// ---- Library/10_Machine/11_IOData/GVL_Output.TcGVL
{attribute 'qualified_only'}
VAR_GLOBAL
	uniDO : uni_OutputModule;
END_VAR

// ---- Library/10_Machine/12_MachineControl/GVL_Machine.TcGVL
VAR_GLOBAL
    PackTags               : ARRAY[0..3] OF ST_PackMLv30; //PackTags
    bButtonProductionReq   : BOOL; //TRUE when a mode change to PRODUCTION is requested
    stChangeIntoProduction : ST_ChangeIntoProduction; //Result of command box "Change to Production requested"
    CylinderStatus         : ST_CylinderStatus;
    RemoteData             : ST_SetupPara;
    AllocatYAxisHome       : BOOL;
END_VAR
VAR_GLOBAL PERSISTENT
    LocalData : ST_SetupPara;
END_VAR

// ---- Library/10_Machine/12_MachineControl/GVL_Machine_Const.TcGVL
VAR_GLOBAL CONSTANT
	udiMax_CylinderNum : UDINT := 53;
END_VAR

// ---- Library/10_Machine/18_HMI_Handshake/GVL_ADS.TcGVL
{attribute 'qualified_only'}
VAR_GLOBAL
	StorageTask 		:   E_MachineTask;
	NeedleTask			:   E_MachineTask;
	ShippingTask		:   E_MachineTask;
	
	PCTask              :  	ST_PCTask;
	//手動模式
	Manualmode			:	ST_MachineAdjust;
	//自動
 	Automode 			:	ST_MachineTask;   
	ActiveFinishing 	:	ST_ActiveResult;
	MachineMode         :   ST_Mode;
	
END_VAR

// ---- Library/10_Machine/18_HMI_Handshake/GVL_HMI.TcGVL
{attribute 'qualified_only'}
VAR_GLOBAL
    ControlOutPut 	: ST_HMI_ControlOutPut;//手臂以及馬達動作命令
    ControlConvery  : ST_HMI_ControlConvery;//軌道動作命令
    ControlInPut 	: ST_HMI_ControlInPut;//X點位
    Setup     		: ST_SetupPara;//參數
    Status    		: ST_HMI_MachineStatus;//狀態
END_VAR

// ---- POUs/ModbusRTU/00_BaseFBs/01_FB_ObjectBase/GVLs/Para_ObjectBase.TcGVL
{attribute 'qualified_only'}
VAR_GLOBAL CONSTANT
	cNumCmdRecord			: UINT := 500;
	cNumMsgRecord			: UINT := 1000;
END_VAR

// ---- Library/00_PackML/01_ObjectBase/I_ErrorElement.TcIO
INTERFACE I_ErrorElement

METHOD M_GetError
VAR_INPUT
END_VAR
VAR_OUTPUT
	Error : BOOL;
	ErrorID : DINT;
	ErrorMsg : T_MaxString;
END_VAR
END_METHOD

METHOD M_GetName :STRING
VAR_INPUT
END_VAR
END_METHOD

METHOD RegisterAlarm
VAR_INPUT
	Trigger : REFERENCE TO BOOL;
	ID : DINT;
	value :DINT;
	Message : STRING;
	Category : DINT;
END_VAR
END_METHOD

END_INTERFACE

// ---- Library/00_PackML/01_ObjectBase/I_ErrorSubject.TcIO
INTERFACE I_ErrorSubject

END_INTERFACE

// ---- POUs/ModbusRTU/00_BaseFBs/01_FB_ObjectBase/ITFs/IBasicElement.TcIO
INTERFACE IBasicElement

METHOD GetModelState
VAR_INPUT
END_VAR
VAR_OUTPUT
    xDone : BOOL;
    xBusy : BOOL;
    xError : BOOL;
    xAborted : BOOL;
    iErrorID : UDINT;
	UniqueErrorCode : STRING;
END_VAR
END_METHOD

METHOD GetName : STRING
VAR_INPUT
END_VAR
END_METHOD

END_INTERFACE

// ---- POUs/ModbusRTU/ComModbusRTU.TcPOU
PROGRAM ComModbusRTU
VAR
	MB_EL6X22B_ControllerN				:	ARRAY[0..3] OF ModbusRtuMasterV2_KL6x22B;
	MBUnusedData_Read 					: 	ARRAY[0..3] OF ARRAY[0..7] OF BYTE;
	MBSensorError_Read 					: 	ARRAY[0..3] OF ARRAY[0..21] OF BYTE;
	nErrID_ControllerN					:	ARRAY[0..3] OF MODBUS_ERRORS;
	iReadMBAddr							:	ARRAY[0..3] OF WORD;
	bBusy_ControllerN					:	ARRAY[0..3] OF BOOL;
	bError_ControllerN					:	ARRAY[0..3] OF BOOL;
	fbComReset_ControllerN				:	ARRAY[0..3] OF ComReset;
	bComReset							:	ARRAY[0..3] OF BOOL;
	bComResetBusy							:	ARRAY[0..3] OF BOOL;
	bComResetError							:	ARRAY[0..3] OF BOOL;
	bStart								:	ARRAY[0..3] OF BOOL;
	
	actStart							:	ARRAY[0..3] OF ULINT;
	actEnd								:	ARRAY[0..3] OF ULINT;
	exeTime								:	ARRAY[0..3] OF ULINT;
	nSlave								:	BYTE;
	MBdata_Read_ControllerN	 AT %I*		: 	ARRAY[0..3] OF ARRAY[0..21] OF BYTE;
	bMasterError						:	ARRAY[0..3] OF BOOL;
	nStep								:	UINT;
	bModbusRTUError						:	BOOL;
	udiModbusRTUErrorID					:	UDINT;
	nAlias								:	UINT;
	bPassModBusMaster					:	ARRAY[0..3] OF BOOL;
	
	
	//================Alternative======================
	//fb_Warehouse_Modbus :ARRAY[0..3] OF FB_CommunicateModbusRTU; //0&1 : warehouse A , 2&3 : warehouse B
		//Declared in GVL due to Error handling request
	I		:UINT;
	SensorState	: ARRAY[0..99] OF BOOL;
	SensorStatesAll : un_RS485States_all;
	arr485sensor					: ARRAY [0..399] OF BOOL;
	fb_Warehouse_Modbus : ARRAY [0..3] OF FB_CommunicateModbusRTU;
	bMotorCoreUpdated	:	BOOL := TRUE;
	bReset				:	BOOL;
END_VAR

//M_CommunicateModbusRTU(bReset:=GVL.Reset,
//						bModBusRTUError=>bModbusRTUError,
//						udiModbusRTUErrorID=>udiModbusRTUErrorID);
						
//GVL.fbModbusRTUErrorTrans(
//	xDone:= , 
//	xBusy:= , 
//	xError:= bModbusRTUError, 
//	xAborted:= , 
//	iErrorID:= udiModbusRTUErrorID, 
//	Name:= 'Communicate ModBus RTU ');
	
	
	
//=================Alternative======================================

//Update FBs
FOR I :=0 TO 3 BY 1 DO
	fb_Warehouse_Modbus[I](Execute:=bMotorCoreUpdated AND NOT bPassModBusMaster[I] , 
							   unitID :=UINT_TO_BYTE(I)+1 , 
							   Reset:=bReset,
							   MBdata_Read_ControllerN :=MBdata_Read_ControllerN[I],
							   ObjectName:=CONCAT('Communicate ModBus RTU : ',UINT_TO_STRING(I)),
							   arrSensor=>SensorStatesAll.arrSensorByController[I]);
	
	arr485sensor := SensorStatesAll.arrSensorAll;
	
END_FOR


//bPassModBusMaster[0] := GVL.stModbusByPass.switchOff_1;
//bPassModBusMaster[1] := GVL.stModbusByPass.switchOff_2;
//bPassModBusMaster[2] := GVL.stModbusByPass.switchOff_3;
//bPassModBusMaster[3] := GVL.stModbusByPass.switchOff_4;

END_PROGRAM

// ---- POUs/ModbusRTU/SerialComTask/FB_CommunicateModbusRTU.TcPOU
FUNCTION_BLOCK FB_CommunicateModbusRTU EXTENDS FB_ObjectBase_V2
VAR_INPUT
//    Execute    :BOOL;   // True : This prog will start.
//    Abort      :BOOL;   // True : This prog will be abort.
//    Reset      :BOOL;   // True : This prog will be reset.
//    ObjectName :STRING; // Set this fb name(About it's action)
	  
	  
	  unitID	  :BYTE;
	  MBdata_Read_ControllerN	: REFERENCE TO 	ARRAY[0..21] OF BYTE;
END_VAR

VAR_OUTPUT
//    Busy    :BOOL;        // True : This prog is running.
//    Done    :BOOL;        // True : Command has been executed.
//    Aborted :BOOL;        // True : This prog is aborted.
//    Error   :BOOL;        // True : This prog has an error.
//    ErrorID :UINT;       // Output ErrorID
//    Status  :T_MaxString; // Output this prog status by string(255bytes)
	arrSensor		: ARRAY[0..99] OF BOOL;
END_VAR

VAR
//    eState :E_MethodStatus_Basic;
//	uiExecutingStep : UDINT; // This var is used to been controll STATE_EXECUTING process.
//	uiResettingStep : UDINT;
//	uiAbortingStep : UDINT;
//	_Executed :BOOL; // Executing process completed.
//	_Error : BOOL; // FB has an error.
//	_ResetCompleted : BOOL; // FB resetting completed.
//	_AbortCompleted : BOOL; // FB aborting completed.
	_Abort		: BOOL;
	strStatus	: STRING;
	uiResumeStep : UINT;
	arrSensorEmpty : ARRAY[0..99] OF BOOL;
	MB_EL6X22B_ControllerN	: ModbusRtuMasterV2_KL6x22B;
	fbComReset_ControllerN	: ComReset;	
	fbClearComBuffer		: ClearComBuffer;
	SensorState : un_RS485States;
	bComReset	:BOOL;
	bComResetBusy :BOOL;
	bComResetError :BOOL;
	bFB_ErrorOccur :BOOL;
END_VAR

A00_BasicUnits();
SUPER^.A10_StateControl();

ACTION A00_BasicUnits:
MB_EL6X22B_ControllerN();
fbComReset_ControllerN(
		Execute:= bComReset, 
		pComIn:= ADR(MB_EL6X22B_ControllerN.InData), 
		pComOut:= ADR(MB_EL6X22B_ControllerN.OutData), 
		SizeComIn:= SIZEOF(MB_EL6X22B_ControllerN.InData), 
		Done=> , 
		Busy=> bComResetBusy, 
		Error=> bComResetError, 
		ErrorID=> );
END_ACTION

METHOD GetModelState
VAR_OUTPUT
    xDone    :BOOL;
    xBusy    :BOOL;
    xError   :BOOL;
    xAborted :BOOL;
    iErrorID :UDINT;
	UniqueErrorCode : STRING;
END_VAR
xDone    := Done;
xBusy    := Busy;
xError   := Error;
xAborted := Abort;
iErrorID := ErrorID;
END_METHOD

METHOD GetName : STRING
GetName := ObjectName;
END_METHOD

METHOD PRIVATE M_AnalyzeData : BOOL
VAR_INPUT
	Data : ARRAY [0..21] OF BYTE;
END_VAR

VAR_OUTPUT
	arrSensor : ARRAY[0..9] OF BOOL;
END_VAR

arrSensor[0] :=Data[4].1;
arrSensor[1] :=Data[4].0;
arrSensor[2] :=Data[3].7;
arrSensor[3] :=Data[3].6;
arrSensor[4] :=Data[3].5;
arrSensor[5] :=Data[3].4;
arrSensor[6] :=Data[3].3;
arrSensor[7] :=Data[3].2;
arrSensor[8] :=Data[3].1;
arrSensor[9] :=Data[3].0;
END_METHOD

METHOD  M_STATE_ABORTED
VAR_INPUT
END_VAR
ERROR :=TRUE;
Busy    := FALSE;
Aborted := TRUE;
Status := strStatus;

IF NOT Execute THEN
	eSTATE:=STATE_RESETTING;
END_IF

IF Execute AND Reset THEN
	uiExecutingStep :=uiResumeStep;
	eSTATE:=STATE_EXECUTING;
END_IF
END_METHOD

METHOD  M_STATE_ABORTING
VAR_INPUT
END_VAR
CASE uiAbortingStep OF
	0 :
		uiAbortingStep:=9999;
	
	9999:	_AbortCompleted:=TRUE;
END_CASE

IF _AbortCompleted THEN	
	eSTATE :=STATE_ABORTED;
END_IF
END_METHOD

METHOD  M_STATE_DONE
VAR_INPUT
END_VAR
Busy 	:= FALSE;
Done	:=TRUE;

IF NOT Execute THEN
	eSTATE:=STATE_RESETTING;
END_IF
END_METHOD

METHOD  M_STATE_DORMANT
VAR_INPUT
END_VAR
Busy            := FALSE;
Done            := FALSE;
Aborted         := FALSE;
Error           := FALSE;
ErrorID         := 0;
Status          := '';
_ResetCompleted := FALSE;
_Error          := FALSE;
_Executed       := FALSE;
strStatus :='No Error';
uiExecutingStep :=uiResettingStep :=uiResumeStep :=0;
bComReset		:= FALSE;

arrSensor :=arrSensorEmpty;
// output all false if program stop working

IF Execute THEN
	eSTATE:=STATE_EXECUTING;
END_IF
END_METHOD

METHOD  M_STATE_ERROR
VAR_INPUT
END_VAR

VAR
	tempStr	:	STRING ;
END_VAR
ERROR   :=TRUE;
Busy	:=FALSE;
tempStr := CONCAT( 'Controllor ' , BYTE_TO_STRING(unitID));
Status := CONCAT(tempStr, strStatus);
ErrorID := unitID + 2600;// Start from 2600

IF NOT Execute OR Reset	THEN	
	eSTATE:=STATE_RESETTING;
END_IF
END_METHOD

METHOD  M_STATE_EXECUTING
VAR_INPUT
END_VAR

VAR
	arrSensorSingleModule : ARRAY [0..9] OF BOOL;	
	pMemoryAddr : ARRAY[0..7] OF BYTE;
END_VAR

VAR_INST
	Quantity : WORD;
	cbLength : UINT;
	
	iReadMBAddr :  WORD :=0;
END_VAR
Busy :=TRUE;
IF  MB_EL6X22B_ControllerN.Error AND NOT bFB_ErrorOccur  THEN
	bFB_ErrorOccur :=TRUE;
	_Error :=TRUE;
	strStatus :=' Modbus connection error';
END_IF

arrSensor:=SensorState.arrSensorByController;

IF iReadMBAddr <= 900 THEN
		Quantity :=10;	
	    cbLength :=20;
		MB_EL6X22B_ControllerN.ReadCoils();
ELSE
		Quantity :=1;
		cbLength :=2;
		MB_EL6X22B_ControllerN.ReadInputRegs();
END_IF

CASE uiExecutingStep OF
	
0: // Init
	MB_EL6X22B_ControllerN.Execute:=FALSE;
	iReadMBAddr:=0;
	uiExecutingStep:=100;
	
100:	
	MB_EL6X22B_ControllerN.UnitID:= unitID;
	MB_EL6X22B_ControllerN.Quantity:= Quantity; 
	MB_EL6X22B_ControllerN.MBAddr:= iReadMBAddr; 
	MB_EL6X22B_ControllerN.cbLength:= cbLength;
	MB_EL6X22B_ControllerN.pMemoryAddr:=ADR(pMemoryAddr) ; 
	MB_EL6X22B_ControllerN.Timeout:= T#1000MS; 
	MB_EL6X22B_ControllerN.Execute:=TRUE;	
	IF MB_EL6X22B_ControllerN.BUSY THEN
		uiExecutingStep:=200;
	END_IF	
	IF bFB_ErrorOccur THEN
		uiExecutingStep:=110;		
	END_IF
	
110:
	bFB_ErrorOccur :=FALSE; //Internal error flag 
	IF MB_EL6X22B_ControllerN.BUSY THEN
		uiExecutingStep:=200;
	END_IF
		
200:
	IF NOT MB_EL6X22B_ControllerN.BUSY THEN
		MB_EL6X22B_ControllerN.Execute:=FALSE;
		
		IF iReadMBAddr>=1000 THEN
			// Error checking step			
			IF MBdata_Read_ControllerN[1] = 4 AND MBdata_Read_ControllerN[3] + MBdata_Read_ControllerN[4] > 0 THEN
				_Error := TRUE;
				strStatus :=' Controller report error';
			END_IF
			
			iReadMBAddr :=0;
			
		ELSE
			// Signal step
			M_AnalyzeData(Data :=MBdata_Read_ControllerN,arrSensor=>arrSensorSingleModule);
			SensorState.arrSensorBySingleModule[iReadMBAddr/100] :=arrSensorSingleModule;		
			iReadMBAddr :=iReadMBAddr +100;
		END_IF
		
		uiExecutingStep:=100;		
		
	 END_IF

END_CASE
	
IF NOT Execute THEN
	eState:=STATE_RESETTING;
END_IF
IF _Error THEN
	eState:=STATE_ERROR;
END_IF
IF _Abort THEN
	eSTATE:=STATE_ABORTING;
END_IF
IF _Executed THEN
	eSTATE:=STATE_Done;
END_IF
END_METHOD

METHOD  M_STATE_RESETTING
VAR_INPUT
END_VAR
Error :=FALSE;
Done :=FALSE;
Busy := FALSE;


CASE uiResettingStep OF
	
	0:
		MB_EL6X22B_ControllerN.Execute:=FALSE;
//		fbClearComBuffer(Buffer:=MB_EL6X22B_ControllerN.InData);
//		fbClearComBuffer(Buffer:=MB_EL6X22B_ControllerN.OutData);
		uiResettingStep:=100;
	100:	
		bComReset := TRUE;
		IF fbComReset_ControllerN.Busy THEN
			uiResettingStep:=200;
		END_IF
	200:
		IF fbComReset_ControllerN.Done THEN
			uiResettingStep:=9999;
		END_IF

	9999:
		_Error:=FALSE;
		_ResetCompleted:=TRUE;
END_CASE
IF _ResetCompleted THEN
	eSTATE:=STATE_DORMANT;
END_IF
END_METHOD

END_FUNCTION_BLOCK

// ---- POUs/ModbusRTU/00_BaseFBs/01_FB_ObjectBase/FB_ObjectBase_V2.TcPOU
FUNCTION_BLOCK FB_ObjectBase_V2 IMPLEMENTS IBasicElement
VAR_INPUT
    Execute    :BOOL;   // True : This prog will start.
    Abort      :BOOL;   // True : This prog will be abort.
    Reset      :BOOL;   // True : This prog will be reset.
    ObjectName :STRING; // Set this fb name(About it's action)
END_VAR

VAR_OUTPUT
    Busy    :BOOL;        // True : This prog is running.
    Done    :BOOL;        // True : Command has been executed.
    Aborted :BOOL;        // True : This prog is aborted.
    Error   :BOOL;        // True : This prog has an error.
    ErrorID :UINT;       // Output ErrorID
    Status  :STRING; // Output this prog status by string(255bytes)
	UniqueErrorCode :STRING;	
END_VAR

VAR
    eState :E_MethodStatus_Basic;
	uiExecutingStep : UDINT; // This var is used to been controll STATE_EXECUTING process.
	uiResettingStep : UDINT;
	uiAbortingStep : UDINT;
	_Executed :BOOL; // Executing process completed.
	_Error : BOOL; // FB has an error.
	_ResetCompleted : BOOL; // FB resetting completed.
	_AbortCompleted : BOOL; // FB aborting completed.
END_VAR

A00_BasicUnits();
A10_StateControl();

ACTION A00_BasicUnits:

END_ACTION

ACTION A10_StateControl:
CASE eState OF
	STATE_DORMANT:
		M_STATE_DORMANT();
	STATE_EXECUTING:
		M_STATE_EXECUTING();
	STATE_ABORTING:
		M_STATE_ABORTING();
	STATE_ABORTED:
		M_STATE_ABORTED();
	STATE_DONE:
		M_STATE_DONE();
	STATE_ERROR:
		M_STATE_ERROR();
	STATE_RESETTING:
		M_STATE_RESETTING();
END_CASE
END_ACTION

METHOD GetModelState
VAR_OUTPUT
    xDone    :BOOL;
    xBusy    :BOOL;
    xError   :BOOL;
    xAborted :BOOL;
    iErrorID :UDINT;	
	UniqueErrorCode : STRING;
END_VAR
xDone    := Done;
xBusy    := Busy;
xError   := Error;
xAborted := Abort;
iErrorID := ErrorID;
UniqueErrorCode := THIS^.UniqueErrorCode;
END_METHOD

METHOD GetName : STRING
GetName := ObjectName;
END_METHOD

METHOD M_RefLinks
VAR_INPUT
END_VAR
END_METHOD

METHOD  M_STATE_ABORTED
VAR_INPUT
END_VAR
;
END_METHOD

METHOD  M_STATE_ABORTING
VAR_INPUT
END_VAR
;
END_METHOD

METHOD  M_STATE_DONE
VAR_INPUT
END_VAR
;
END_METHOD

METHOD  M_STATE_DORMANT
VAR_INPUT
END_VAR
;
END_METHOD

METHOD  M_STATE_ERROR
VAR_INPUT
END_VAR
;
END_METHOD

METHOD  M_STATE_EXECUTING
VAR_INPUT
END_VAR
;
END_METHOD

METHOD  M_STATE_RESETTING
VAR_INPUT
END_VAR
;
END_METHOD

END_FUNCTION_BLOCK

// ---- POUs/DAS_CoreSys.TcPOU
PROGRAM DAS_CoreSys
VAR
    UserModeCofig  : PML_UnitModeConfig; //User can configure his own Mode
    MachineControl : FB_MachineControl;
	CoreSys_Stop : BOOL;
	CoreSys_Reset :BOOL;
	CoreSys_Start : BOOL;
	CoreSys_Estop : BOOL;
	OP_Mode : E_UnitMode := E_UnitMode.Manual;
END_VAR

A00_BasicUnit();
A10_StatusCtrl();


CASE GVL_ADS.MachineMode.TargetMode OF
		E_MachineMode.MANUAL:
			OP_Mode := E_UnitMode.Manual;
		E_MachineMode.AUTO:
			OP_Mode := E_UnitMode.Auto;
ELSE
	OP_Mode := E_UnitMode.Manual;
END_CASE
IF OP_Mode = E_UnitMode.Manual THEN
	GVL_ADS.MachineMode.CurrentMode := E_MachineMode.MANUAL;
ELSIF OP_Mode = E_UnitMode.Auto THEN
	GVL_ADS.MachineMode.CurrentMode := E_MachineMode.AUTO;
END_IF

ACTION A00_BasicUnit:
CoreSys_Start := MachineControl.Machine_Start;
CoreSys_Stop := MachineControl.Machine_Stop;
CoreSys_Reset := MachineControl.Machine_Reset;
MachineControl(
    eModeCommand := PackTags[0].Command.UnitMode,
    eStateCommand := PackTags[0].Command.CntrlCmd,
    PackTag := PackTags[0],
    INPUT := GVL_Input.uniDI.stDI,
    OUTPUT := GVL_Output.uniDO.stDO); // FB_MachineControl
PackTags[0].Status.StateCurrent := MachineControl.eStateCurrent;
PackTags[0].Status.UnitModeCurrent := MachineControl.eModeCurrent;
CoreSys_Estop := MachineControl.Machine_Estop;
END_ACTION

ACTION A01_UnitModeConfig:
//UserModeCofig(
//	eMode							:= ePMLUnitMode_Service, 
//	bDisableClearing				:= TRUE, 
//	bDisableStarting				:= TRUE, 
//	bDisableSuspended				:= FALSE, 
//	bDisableStopping				:= TRUE, 
//	bDisableAborting				:= TRUE, 
//	bDisableHolding					:= TRUE, 
//	bDisableHeld					:= TRUE, 
//	bDisableUnholding				:= TRUE, 
//	bDisableSuspending				:= TRUE, 
//	bDisableUnsuspending			:= TRUE, 
//	bDisableResetting				:= TRUE, 
//	bDisableIdle					:= TRUE, 
//	bDisableCompleting				:= TRUE, 
//	bDisableComplete				:= TRUE, 
//	bEnableUnitModeChangeStopped	:= TRUE, 
//	bEnableUnitModeChangeIdle		:= FALSE, 
//	bEnableUnitModeChangeSuspended	:= FALSE, 
//	bEnableUnitModeChangeExecute	:= FALSE, 
//	bEnableUnitModeChangeAborted	:= TRUE, 
//	bEnableUnitModeChangeHeld		:= FALSE, 
//	bEnableUnitModeChangeComplete	:= FALSE, 
//	bError							=> , 
//	nErrorId						=> );
END_ACTION

ACTION A10_StatusCtrl:
IF PackTags[0].Status.UnitModeCurrent = E_UnitMode.Manual THEN
	IF PackTags[0].Status.StateCurrent = ePMLState_Aborted AND NOT MachineControl.Error THEN
		PackTags[0].Command.CntrlCmd := ePMLCommand_Clear;
	END_IF
	IF PackTags[0].Status.StateCurrent = ePMLState_Stopped THEN
		IF OP_Mode = E_UnitMode.Manual THEN
		PackTags[0].Command.CntrlCmd := ePMLCommand_Reset;
		END_IF
	END_IF
	IF PackTags[0].Status.StateCurrent = ePMLState_Idle THEN
		PackTags[0].Command.CntrlCmd := ePMLCommand_Start;
	END_IF
ELSIF PackTags[0].Status.UnitModeCurrent = E_UnitMode.Auto THEN
	IF PackTags[0].Status.StateCurrent = ePMLState_Aborted AND NOT MachineControl.Error THEN
		PackTags[0].Command.CntrlCmd := ePMLCommand_Clear;
	END_IF
	IF PackTags[0].Status.StateCurrent = ePMLState_Stopped THEN
		IF OP_Mode = E_UnitMode.Auto THEN
		PackTags[0].Command.CntrlCmd := ePMLCommand_Reset;
		END_IF
	END_IF
	IF PackTags[0].Status.StateCurrent = ePMLState_Idle THEN
		PackTags[0].Command.CntrlCmd := ePMLCommand_Start;
	END_IF
END_IF

IF PackTags[0].Status.UnitModeCurrent = E_UnitMode.Manual THEN
    IF ((PackTags[0].Status.StateCurrent = ePMLState_Stopped) OR
        (PackTags[0].Status.StateCurrent = ePMLState_Aborted) OR
        (PackTags[0].Status.StateCurrent = ePMLState_Execute)) AND
        MachineControl.MachineHomed
        THEN
        IF OP_Mode = E_UnitMode.Auto THEN
            PackTags[0].Command.UnitMode := E_UnitMode.Auto;
			IF PackTags[0].Status.StateCurrent = ePMLState_Execute THEN
				PackTags[0].Command.CntrlCmd := ePMLCommand_Stop;
			END_IF
        END_IF
    END_IF
ELSIF PackTags[0].Status.UnitModeCurrent = E_UnitMode.Auto THEN
    IF ((PackTags[0].Status.StateCurrent = ePMLState_Stopped) OR
        (PackTags[0].Status.StateCurrent = ePMLState_Aborted) OR
        (PackTags[0].Status.StateCurrent = ePMLState_Execute))
        THEN
        IF OP_Mode = E_UnitMode.Manual THEN
			IF PackTags[0].Status.StateCurrent <> ePMLState_Aborted OR PackTags[0].Status.StateCurrent <> ePMLState_Aborting THEN
				PackTags[0].Command.CntrlCmd := ePMLCommand_Abort;
			END_IF
            PackTags[0].Command.UnitMode := E_UnitMode.Manual;
        END_IF
    END_IF
END_IF

GVL_ADS.OpPannel_Status.EStopBtnStatus := CoreSys_Estop;
GVL_ADS.OpPannel_Status.ResetBtnStatus := CoreSys_Reset;
GVL_ADS.OpPannel_Status.StartBtnStatus := CoreSys_Start;
GVL_ADS.OpPannel_Status.StopBtnStatus := CoreSys_Stop;
// Start
IF PackTags[0].Status.UnitModeCurrent = E_UnitMode.Auto THEN
	CASE PackTags[0].Status.StateCurrent OF
		ePMLState_Idle:
			IF CoreSys_Start THEN
				PackTags[0].Command.CntrlCmd := ePMLCommand_Start;
			END_IF
	END_CASE
END_IF

// Reset & Clear

IF PackTags[0].Status.UnitModeCurrent = E_UnitMode.Auto THEN
	CASE PackTags[0].Status.StateCurrent OF
		ePMLState_Stopped,ePMLState_Complete:
			IF CoreSys_Reset THEN
				PackTags[0].Command.CntrlCmd := ePMLCommand_Reset;
			END_IF
		ePMLState_Aborted:
			IF CoreSys_Reset THEN
				PackTags[0].Command.CntrlCmd := ePMLCommand_Clear;
			END_IF
		ePMLState_Held:
			IF CoreSys_Reset THEN
				PackTags[0].Command.CntrlCmd := ePMLCommand_Unhold;
			END_IF
		ePMLState_Suspended:
			IF CoreSys_Reset THEN
				PackTags[0].Command.CntrlCmd := ePMLCommand_Unsuspend;
			END_IF
	END_CASE
END_IF

// Stop

//IF PackTags[0].Status.UnitModeCurrent = E_UnitMode.Auto THEN
//	CASE PackTags[0].Status.StateCurrent OF
//		ePMLState_Execute:
//			IF CoreSys_Stop THEN
//				PackTags[0].Command.CntrlCmd := ePMLCommand_Suspend;
//			END_IF
//	END_CASE
//END_IF
END_ACTION

END_PROGRAM

// ---- Library/10_Machine/12_MachineControl/FB_MachineControl.TcPOU
FUNCTION_BLOCK FB_MachineControl EXTENDS FB_ModeBase_V2 IMPLEMENTS I_UnitState
VAR_INPUT
    INPUT            : REFERENCE TO ST_InputTable;
    OUTPUT           : REFERENCE TO ST_OutputTable;
    EnableSimulation : BOOL       := FALSE	;
    DataDirect       : E_DataFrom := E_DataFrom.Remote;
END_VAR
VAR_OUTPUT
    Error               : BOOL;
    ErrorID             : DINT;
    ErrMsg              : T_MaxString;
    CylinderStatus      : ST_CylinderStatus;
    MotorStatus         : ST_MotorStatus;
    StorageRobot_EStop  : BOOL;
    ShippingRobot_EStop : BOOL;
    MachineHomed        : BOOL;
    // Machine OpPannel 
    Machine_Estop : BOOL;
    Machine_Start : BOOL;
    Machine_Stop  : BOOL;
    Machine_Reset : BOOL;
END_VAR
VAR
    // C# HMI handshake
    fbHmiHandShakeController : FB_HmiHandShake;

    // internal Output
    InternalOutput : ST_OutputTable;

    // Componets setup parameter
    CurrentData : ST_SetupPara;

    // Current Manual Command
    AllocateManualCommand   : ST_Manual_Allocated;
    StorageManualCommand    : ST_Manual_Storage;
    ShippingManualCommand   : ST_Manual_Shipping;
    AllocateHalfAutoCommand : REFERENCE TO ST_HalfAuto_Allocated;
    // Area controller
    fbAllocateArea : FB_AllocateAreaWithRoundbelt;
    fbStorageArea  : FB_StorageArea;
    fbShippingArea : FB_ShippingArea;

    // Service controller
    TableMove : FB_TableMove;
	fbMachineHoming : FB_MachineHoming;
    // Componets
    Cylinder           : UNI_CylinderList;
    Motor              : UNI_MotorList;
    FanucRobot         : UNI_FanucRobotList;
    CylinderManualCtrl : ARRAY[1..53] OF FB_CylinderManualCtrl;
	MotorManualCtrl    : ARRAY[1..26] OF 	FB_MotorManualCtrl;
    // Wheelhouse Sensor
    WheelhouseSensor : UNI_HMI_WheelHouseInput;

    bCheckMotorWork   : BOOL;
    Service_Handshake : ST_HMI_Handshake; // To read legacy HMI data
    StorageService    : ST_StorageService;
    AllocateService   : ST_AllocateService;
    ShippingService   : ST_ShippingService;
	
    Allocate_EStop			: BOOL;
    Storage_EStop  			: BOOL;
	Allocate_EStopEdgeDetect : FB_EdgeDetect;
    Storage_EstopEdgeDetect  : FB_EdgeDetect;
	
	bStorage_AirPressure 	: BOOL;
	// ErrorHandler
	fbErrorHandler 		:FB_ErrorHandler;
	ErrorTableInitDone 	: BOOL;
	E_StopEdgeDetect	: FB_EdgeDetect;
	StartEdgeDetect 	: FB_EdgeDetect;
	ResetEdgeDetect 	: FB_EdgeDetect;
	StopEdgeDetect 		: FB_EdgeDetect;
	bSafetyDoorOpen 	: BOOL;
	fbBlink_05 			: BLINK;
	bStopMem 			: BOOL;
    fb_AllocateSignalTower : FB_SignalTower;
    fb_StorageSignalTower  : FB_SignalTower;
	_RedLamp 			: BOOL;
	_YellowLamp			: BOOL;
	_GreenLamp 			: BOOL;
	_Buzz 				: BOOL;
	bTest2 				: BOOL;
	
	//Btn ctrl
	tofResetDelay	:TOF;
	tofStopDelay	:TOF;
	tofStartDelay	:TOF;
	
	tonDelayErrorHandle : TON;
END_VAR

// Implement PackML State Machine
SUPER^();
tonDelayErrorHandle(IN:=TRUE, PT:=T#5S); // Delay 5s after PLC run then check error
A00_BaseUnits();
A01_Cylinder();
A02_Motor();
A03_FanucRobot();
A04_OpPannel();
A05_Light();
IF tonDelayErrorHandle.Q THEN
	A10_ErrorHandler();
END_IF

IF NOT EnableSimulation THEN
    OUTPUT := InternalOutput;
ELSE
    M_ClearOutput();
END_IF

WheelhouseSensor.arWheelHouseInput := ComModbusRTU.arr485sensor;

IF DataDirect = E_DataFrom.Local THEN
    CurrentData := GVL_Machine.LocalData;
ELSIF DataDirect = E_DataFrom.Remote THEN
    CurrentData := GVL_Machine.RemoteData;
    AllocateManualCommand := GVL_HMI.Allocated.Manual;
    StorageManualCommand := GVL_HMI.Storage.Manual;
    ShippingManualCOmmand := GVL_HMI.Shipping.Manual;
    AllocateHalfAutoCommand REF= GVL_HMI.Allocated.HalfAuto;
END_IF
gvl_ads.MachineState := FUN_MachineState(
	Error:= xError, 
	Estop:= FALSE, 
	Stop:= Machine_Stop, 
	Reset:= Machine_Reset OR tofResetDelay.Q , 
	Start:= Machine_Start,
	eMachineState :=  gvl_ads.MachineState,
	HomeBusy:= fbMachineHoming.xBusy, 
	Homed:= MachineHomed, 
	MachineMode:= eModeCurrent);

ACTION A00_BaseUnits:
fbStorageArea(eModeCommand :=,
              eStateCommand :=,
			  FanucRobot := FanucRobot.List.StorageRobot,
              PackTag := GVL_Machine.PackTags[UnitNo.Storage],
			  Service := StorageService,
			  WheelhouseSensor :=WheelhouseSensor,
			  Motor := Motor,
			  Input := INPUT,
			  Output := InternalOutput,
			  Reset := Machine_Reset,
			  Stop := Machine_Stop,
			  bStopMem:=bStopMem,
			  Cylinder:= Cylinder,
			  CurrentData :=CurrentData,
              eModeCurrent => GVL_Machine.PackTags[UnitNo.Storage].Status.UnitModeCurrent,
              eStateCurrent => GVL_Machine.PackTags[UnitNo.Storage].Status.StateCurrent);

fbAllocateArea(eModeCommand :=,
               eStateCommand :=,
			   INPUT :=INPUT,
			   OUTPUT :=InternalOutput,
			   Cylinder := Cylinder,
			   Motor := Motor,
			   Reset := Machine_Reset,
			   Stop := Machine_Stop,
			   bStopMem:=bStopMem,
			   CurrentData := CurrentData,
               PackTag := GVL_Machine.PackTags[UnitNo.Allocate],
			   service := AllocateService,
               eModeCurrent => GVL_Machine.PackTags[UnitNo.Allocate].Status.UnitModeCurrent,
               eStateCurrent => GVL_Machine.PackTags[UnitNo.Allocate].Status.StateCurrent);

fbShippingArea(eModeCommand :=,
               eStateCommand :=,
			   FanucRobot:= FanucRobot.List.ShippingRobot,
			   INPUT :=INPUT,
			   Motor := Motor,
			   Reset := Machine_Reset,
			   Stop := Machine_Stop,
			   bStopMem:=bStopMem,
               PackTag := GVL_Machine.PackTags[UnitNo.Shipping],
			   Service := ShippingService,
               eModeCurrent => GVL_Machine.PackTags[UnitNo.Shipping].Status.UnitModeCurrent,
               eStateCurrent => GVL_Machine.PackTags[UnitNo.Shipping].Status.StateCurrent);

fbHmiHandShakeController(xEnable := TRUE,CylinderStatus := CylinderStatus,MotorStatus:=MotorStatus,FanucRobot := FanucRobot);

fbMachineHoming(
	xDone=> , 
	xBusy=> , 
	xError=> , 
	xExecute:= , 
	xAbort:= , 
	AllocateHome:= fbAllocateArea.fbAllocateHome, 
	StorageHome:= fbStorageArea.fbStorageHoming, 
	ShippingHome:= fbShippingArea.fbShippingHoming, 
	AllocateHomed:= fbAllocateArea.Homed, 
	StorageHomed:= fbStorageArea.Homed, 
	ShippingHomed:= fbShippingArea.Homed, 
	Homed:= MachineHomed, 
	TimeOut:= , 
	xAborted=> , 
	iErrorID=> , 
	ErrorMsg=> );
	
fbErrorHandler(
	xDone=> , 
	xBusy=> , 
	xError=> , 
	AlarmList:= PackTag.Admin.Alarm,
	AlarmHistory := PackTag.Admin.AlarmHistory, 
	HMI_AlarmMonitorList:= GVL_ADS.AlarmAllocation, 
	MaxRecords:= 1000, 
	ResetAllAlarms:= ,
	Reset := Machine_Reset OR tofResetDelay.Q , 
	EnableLogging:= , 
	ActiveAlarmCount=> , 
	TotalRecords=> , 
	SystemStatus=> );
	
fbBlink_05(ENABLE:= TRUE, TIMELOW:= T#0.25S, TIMEHIGH:= T#0.25S, OUT=> );
Allocate_EStopEdgeDetect(xInput := INPUT.bAllocate_EStopPb);
Storage_EstopEdgeDetect(xInput := INPUT.bStorage_EstopPb);
END_ACTION

ACTION A01_Cylinder:
cylinder.List.fbUpCV_FeedInPress1(xDone =>,
                                  xBusy =>,
                                  xError =>CylinderStatus.UpCV_FeedInPress1.Error,
                                  xEnable :=,
                                  FrontSensor :=,
                                  RearSensor :=,
                                  SetupPara := CurrentData.Cylinders.UpCV_FeedInPress1,
                                  CurrentCylinderType =>,
                                  InFrontPosition => CylinderStatus.UpCV_FeedInPress1.InFrontPosition,
                                  InRearPosition =>CylinderStatus.UpCV_FeedInPress1.InRearPosition,
                                  ExtendOutput => InternalOutput.bUpCV_FeedInPress1_Valve,
                                  RetractOutput =>);

cylinder.List.fbUpCV_FeedInPress2(xDone =>,
                                  xBusy =>,
                                  xError =>CylinderStatus.UpCV_FeedInPress2.Error,
                                  xEnable :=,
                                  FrontSensor :=,
                                  RearSensor :=,
                                  SetupPara := CurrentData.Cylinders.UpCV_FeedInPress2,
                                  CurrentCylinderType =>,
                                  InFrontPosition =>CylinderStatus.UpCV_FeedInPress2.InFrontPosition,
                                  InRearPosition =>CylinderStatus.UpCV_FeedInPress2.InRearPosition,
                                  ExtendOutput => InternalOutput.bUpCV_FeedInPress2_Valve,
                                  RetractOutput =>);

cylinder.List.fbUpCV_DiameterPress(xDone =>,
                                   xBusy =>,
                                   xError =>CylinderStatus.UpCV_DiameterPress.Error,
                                   xEnable :=,
                                   FrontSensor :=,
                                   RearSensor :=,
                                   SetupPara := CurrentData.Cylinders.UpCV_DiameterPress,
                                   CurrentCylinderType =>,
                                   InFrontPosition =>CylinderStatus.UpCV_DiameterPress.InFrontPosition,
                                   InRearPosition =>CylinderStatus.UpCV_DiameterPress.InRearPosition,
                                   ExtendOutput => InternalOutput.bUpCV_DiameterPress_Valve,
                                   RetractOutput =>);

cylinder.List.fbUpCV_CamaraPress1(xDone =>,
                                  xBusy =>,
                                  xError =>CylinderStatus.UpCV_CamaraPress1.Error,
                                  xEnable :=,
                                  FrontSensor :=,
                                  RearSensor :=,
                                  SetupPara := CurrentData.Cylinders.UpCV_CamaraPress1,
                                  CurrentCylinderType =>,
                                  InFrontPosition =>CylinderStatus.UpCV_CamaraPress1.InFrontPosition,
                                  InRearPosition =>CylinderStatus.UpCV_CamaraPress1.InRearPosition,
                                  ExtendOutput => InternalOutput.bUpCV_CamaraPress1_Valve,
                                  RetractOutput =>);

cylinder.List.fbUpCV_CamaraPress2(xDone =>,
                                  xBusy =>,
                                  xError =>CylinderStatus.UpCV_CamaraPress2.Error,
                                  xEnable :=,
                                  FrontSensor :=,
                                  RearSensor :=,
                                  SetupPara := CurrentData.Cylinders.UpCV_CamaraPress2,
                                  CurrentCylinderType =>,
                                  InFrontPosition =>CylinderStatus.UpCV_CamaraPress2.InFrontPosition,
                                  InRearPosition =>CylinderStatus.UpCV_CamaraPress2.InRearPosition,
                                  ExtendOutput => InternalOutput.bUpCV_CamaraPress2_Valve,
                                  RetractOutput =>);

cylinder.List.fbUpCV_CamaraPress3(xDone =>,
                                  xBusy =>,
                                  xError =>CylinderStatus.UpCV_CamaraPress3.Error,
                                  xEnable :=,
                                  FrontSensor :=,
                                  RearSensor :=,
                                  SetupPara := CurrentData.Cylinders.UpCV_CamaraPress3,
                                  CurrentCylinderType =>,
                                  InFrontPosition =>CylinderStatus.UpCV_CamaraPress3.InFrontPosition,
                                  InRearPosition =>CylinderStatus.UpCV_CamaraPress3.InRearPosition,
                                  ExtendOutput => InternalOutput.bUpCV_CamaraPress3_Valve,
                                  RetractOutput =>);

cylinder.List.fbUpCV_CamaraPress4(xDone =>, 
                                  xBusy =>,
                                  xError =>CylinderStatus.UpCV_CamaraPress4.Error,
                                  xEnable :=,
                                  FrontSensor :=,
                                  RearSensor :=,
                                  SetupPara := CurrentData.Cylinders.UpCV_CamaraPress4,
                                  CurrentCylinderType =>,
                                  InFrontPosition =>CylinderStatus.UpCV_CamaraPress4.InFrontPosition,
                                  InRearPosition =>CylinderStatus.UpCV_CamaraPress4.InRearPosition,
                                  ExtendOutput => InternalOutput.bUpCV_CamaraPress4_Valve,
                                  RetractOutput =>);

cylinder.List.fbUpCV_Block1(xDone =>,
                            xBusy =>,
                            xError =>CylinderStatus.UpCV_Block1.Error,
                            xEnable :=,
                            FrontSensor :=,
                            RearSensor := INPUT.bUpCV_Block1_RearSensor,
                            SetupPara := CurrentData.Cylinders.UpCV_Block1,
                            CurrentCylinderType =>,
                            InFrontPosition =>CylinderStatus.UpCV_Block1.InFrontPosition,
                            InRearPosition =>CylinderStatus.UpCV_Block1.InRearPosition,
                            ExtendOutput => InternalOutput.bUpCV_Block1_Up_Valve,
                            RetractOutput => InternalOutput.bUpCV_Block1_Down_Valve);
cylinder.List.fbUpCV_Block1.IsDoubleValve := TRUE;

cylinder.List.fbUpCV_Block2(xDone =>,
                            xBusy =>,
                            xError =>CylinderStatus.UpCV_Block2.Error,
                            xEnable :=,
                            FrontSensor :=,
                            RearSensor := INPUT.bUpCV_Block2_RearSensor,
                            SetupPara := CurrentData.Cylinders.UpCV_Block2,
                            CurrentCylinderType =>,
                            InFrontPosition =>CylinderStatus.UpCV_Block2.InFrontPosition,
                            InRearPosition =>CylinderStatus.UpCV_Block2.InRearPosition,
                            ExtendOutput => InternalOutput.bUpCV_Block2_Up_Valve,
                            RetractOutput => InternalOutput.bUpCV_Block2_Down_Valve);
cylinder.List.fbUpCV_Block2.IsDoubleValve := TRUE;

cylinder.List.fbUpCV_Block3(xDone =>,
                            xBusy =>,
                            xError =>CylinderStatus.UpCV_Block3.Error,
                            xEnable :=,
                            FrontSensor :=,
                            RearSensor := INPUT.bUpCV_Block3_RearSensor,
                            SetupPara := CurrentData.Cylinders.UpCV_Block3,
                            CurrentCylinderType =>,
                            InFrontPosition =>CylinderStatus.UpCV_Block3.InFrontPosition,
                            InRearPosition =>CylinderStatus.UpCV_Block3.InRearPosition,
                            ExtendOutput => InternalOutput.bUpCV_Block3_Up_Valve,
                            RetractOutput => InternalOutput.bUpCV_Block3_Down_Valve);
cylinder.List.fbUpCV_Block3.IsDoubleValve := TRUE;

cylinder.List.fbUpCV_DiameterHoriz(xDone =>,
                                   xBusy =>,
                                   xError =>CylinderStatus.UpCV_DiameterHoriz.Error,
                                   xEnable :=,
                                   FrontSensor := INPUT.bUpCV_DiameterHoriz_FrontSensor,
                                   RearSensor := INPUT.bUpCV_DiameterHoriz_RearSensor,
                                   SetupPara := CurrentData.Cylinders.UpCV_DiameterHoriz,
                                   CurrentCylinderType =>,
                                   InFrontPosition =>CylinderStatus.UpCV_DiameterHoriz.InFrontPosition,
                                   InRearPosition =>CylinderStatus.UpCV_DiameterHoriz.InRearPosition,
                                   ExtendOutput => InternalOutput.bUpCV_DiameterHoriz_Extend_Valve,
                                   RetractOutput => InternalOutput.bUpCV_DiameterHoriz_Retract_Valve);
cylinder.List.fbUpCV_DiameterHoriz.IsDoubleValve := TRUE;

cylinder.List.fbUpCV_DiameterVert(xDone =>,
                                  xBusy =>,
                                  xError =>CylinderStatus.UpCV_DiameterVert.Error,
                                  xEnable :=,
                                  FrontSensor := INPUT.bUpCV_DiameterVert_FrontSensor,
                                  RearSensor := INPUT.bUpCV_DiameterVert_RearSensor,
                                  SetupPara := CurrentData.Cylinders.UpCV_DiameterVert,
                                  CurrentCylinderType =>,
                                  InFrontPosition =>CylinderStatus.UpCV_DiameterVert.InFrontPosition,
                                  InRearPosition =>CylinderStatus.UpCV_DiameterVert.InRearPosition,
                                  ExtendOutput => InternalOutput.bUpCV_DiameterVert_Valve,
                                  RetractOutput =>);

cylinder.List.fbUpCV_DiameterClamp(xDone =>,
                                   xBusy =>,
                                   xError =>CylinderStatus.UpCV_DiameterClamp.Error,
                                   xEnable :=,
                                   FrontSensor :=,
                                   RearSensor :=,
                                   SetupPara := CurrentData.Cylinders.UpCV_DiameterClamp,
                                   CurrentCylinderType =>,
                                   InFrontPosition =>CylinderStatus.UpCV_DiameterClamp.InFrontPosition,
                                   InRearPosition =>CylinderStatus.UpCV_DiameterClamp.InRearPosition,
                                   ExtendOutput => InternalOutput.bUpCV_DiameterClamp_Close_Valve,
                                   RetractOutput => InternalOutput.bUpCV_DiameterClamp_Open_Valve);
cylinder.List.fbUpCV_DiameterClamp.IsDoubleValve := TRUE;

cylinder.List.fbStackPush(xDone =>,
                          xBusy =>,
                          xError =>CylinderStatus.StackPush.Error,
                          xEnable :=,
                          FrontSensor := INPUT.bStackPush_Pusher_FrontSensor,
                          RearSensor := INPUT.bStackPush_Pusher_RearSensor,
                          SetupPara := CurrentData.Cylinders.StackPush,
                          CurrentCylinderType =>,
                          InFrontPosition =>CylinderStatus.StackPush.InFrontPosition,
                          InRearPosition =>CylinderStatus.StackPush.InRearPosition,
                          ExtendOutput => InternalOutput.bStackPush_Valve,
                          RetractOutput =>);

cylinder.List.fbPullOutCV_AsidePress1(xDone =>,
                                      xBusy =>,
                                      xError =>CylinderStatus.PullOutCV_AsidePress1.Error,
                                      xEnable :=,
                                      FrontSensor :=,
                                      RearSensor :=,
                                      SetupPara := CurrentData.Cylinders.PullOutCV_AsidePress1,
                                      CurrentCylinderType =>,
                                      InFrontPosition =>CylinderStatus.PullOutCV_AsidePress1.InFrontPosition,
                                      InRearPosition =>CylinderStatus.PullOutCV_AsidePress1.InRearPosition,
                                      ExtendOutput => InternalOutput.bPullOutCV_AsidePress1_Valve,
                                      RetractOutput =>);

cylinder.List.fbPullOutCV_AsidePress2(xDone =>,
                                      xBusy =>,
                                      xError =>CylinderStatus.PullOutCV_AsidePress2.Error,
                                      xEnable :=,
                                      FrontSensor :=,
                                      RearSensor :=,
                                      SetupPara := CurrentData.Cylinders.PullOutCV_AsidePress2,
                                      CurrentCylinderType =>,
                                      InFrontPosition =>CylinderStatus.PullOutCV_AsidePress2.InFrontPosition,
                                      InRearPosition =>CylinderStatus.PullOutCV_AsidePress2.InRearPosition,
                                      ExtendOutput => InternalOutput.bPullOutCV_AsidePress2_Valve,
                                      RetractOutput =>);

cylinder.List.fbPullOutCV_AsideBlock(xDone =>,
                                     xBusy =>,
                                     xError =>CylinderStatus.PullOutCV_AsideBlock.Error,
                                     xEnable :=,
                                     FrontSensor :=,
                                     RearSensor := INPUT.bPullOutCV_AsideBlock_RearSensor,
                                     SetupPara := CurrentData.Cylinders.PullOutCV_AsideBlock,
                                     CurrentCylinderType =>,
                                     InFrontPosition =>CylinderStatus.PullOutCV_AsideBlock.InFrontPosition,
                                     InRearPosition =>CylinderStatus.PullOutCV_AsideBlock.InRearPosition,
                                     ExtendOutput => InternalOutput.bPullOutCV_AsideBlock_Valve,
                                     RetractOutput =>);

cylinder.List.fbPullOutCV_BsidePress1(xDone =>,
                                      xBusy =>,
                                      xError =>CylinderStatus.PullOutCV_BsidePress1.Error,
                                      xEnable :=,
                                      FrontSensor :=,
                                      RearSensor :=,
                                      SetupPara := CurrentData.Cylinders.PullOutCV_BsidePress1,
                                      CurrentCylinderType =>,
                                      InFrontPosition =>CylinderStatus.PullOutCV_BsidePress1.InFrontPosition,
                                      InRearPosition =>CylinderStatus.PullOutCV_BsidePress1.InRearPosition,
                                      ExtendOutput => InternalOutput.bPullOutCV_BsidePress1_Valve,
                                      RetractOutput =>);

cylinder.List.fbPullOutCV_BsidePress2(xDone =>,
                                      xBusy =>,
                                      xError =>CylinderStatus.PullOutCV_BsidePress2.Error,
                                      xEnable :=,
                                      FrontSensor :=,
                                      RearSensor :=,
                                      SetupPara := CurrentData.Cylinders.PullOutCV_BsidePress2,
                                      CurrentCylinderType =>,
                                      InFrontPosition =>CylinderStatus.PullOutCV_BsidePress2.InFrontPosition,
                                      InRearPosition =>CylinderStatus.PullOutCV_BsidePress2.InRearPosition,
                                      ExtendOutput => InternalOutput.bPullOutCV_BsidePress2_Valve,
                                      RetractOutput =>);

cylinder.List.fbPullOutCV_BsideBlock(xDone =>,
                                     xBusy =>,
                                     xError =>CylinderStatus.PullOutCV_BsideBlock.Error,
                                     xEnable :=,
                                     FrontSensor :=,
                                     RearSensor := INPUT.bPullOutCV_BsideBlock_RearSensor,
                                     SetupPara := CurrentData.Cylinders.PullOutCV_BsideBlock,
                                     CurrentCylinderType =>,
                                     InFrontPosition =>CylinderStatus.PullOutCV_BsideBlock.InFrontPosition,
                                     InRearPosition =>CylinderStatus.PullOutCV_BsideBlock.InRearPosition,
                                     ExtendOutput => InternalOutput.bPullOutCV_BsideBlock_Valve,
                                     RetractOutput =>);

cylinder.List.fbLowCV_Press1(xDone =>,
                             xBusy =>,
                             xError =>CylinderStatus.LowCV_Press1.Error,
                             xEnable :=,
                             FrontSensor :=,
                             RearSensor :=,
                             SetupPara := CurrentData.Cylinders.LowCV_Press1,
                             CurrentCylinderType =>,
                             InFrontPosition =>CylinderStatus.LowCV_Press1.InFrontPosition,
                             InRearPosition =>CylinderStatus.LowCV_Press1.InRearPosition,
                             ExtendOutput => InternalOutput.bLowCV_Press1_Valve,
                             RetractOutput =>);

cylinder.List.fbLowCV_Press2(xDone =>,
                             xBusy =>,
                             xError =>CylinderStatus.LowCV_Press2.Error,
                             xEnable :=,
                             FrontSensor :=,
                             RearSensor :=,
                             SetupPara := CurrentData.Cylinders.LowCV_Press2,
                             CurrentCylinderType =>,
                             InFrontPosition =>CylinderStatus.LowCV_Press2.InFrontPosition,
                             InRearPosition =>CylinderStatus.LowCV_Press2.InRearPosition,
                             ExtendOutput => InternalOutput.bLowCV_Press2_Valve,
                             RetractOutput =>);

cylinder.List.fbLowCV_Press3(xDone =>,
                             xBusy =>,
                             xError =>CylinderStatus.LowCV_Press3.Error,
                             xEnable :=,
                             FrontSensor :=,
                             RearSensor :=,
                             SetupPara := CurrentData.Cylinders.LowCV_Press3,
                             CurrentCylinderType =>,
                             InFrontPosition =>CylinderStatus.LowCV_Press3.InFrontPosition,
                             InRearPosition =>CylinderStatus.LowCV_Press3.InRearPosition,
                             ExtendOutput => InternalOutput.bLowCV_Press3_Valve,
                             RetractOutput =>);

cylinder.List.fbLowCV_Press4(xDone =>,
                             xBusy =>,
                             xError =>CylinderStatus.LowCV_Press4.Error,
                             xEnable :=,
                             FrontSensor :=,
                             RearSensor :=,
                             SetupPara := CurrentData.Cylinders.LowCV_Press4,
                             CurrentCylinderType =>,
                             InFrontPosition =>CylinderStatus.LowCV_Press4.InFrontPosition,
                             InRearPosition =>CylinderStatus.LowCV_Press4.InRearPosition,
                             ExtendOutput => InternalOutput.bLowCV_Press4_Valve,
                             RetractOutput =>);

cylinder.List.fbLowCV_Block1(xDone =>,
                             xBusy =>,
                             xError =>CylinderStatus.LowCV_Block1.Error,
                             xEnable :=,
                             FrontSensor :=,
                             RearSensor := INPUT.bLowCV_Block1_RearSensor,
                             SetupPara := CurrentData.Cylinders.LowCV_Block1,
                             CurrentCylinderType =>,
                             InFrontPosition =>CylinderStatus.LowCV_Block1.InFrontPosition,
                             InRearPosition =>CylinderStatus.LowCV_Block1.InRearPosition,
                             ExtendOutput => InternalOutput.bLowCV_Block1_Down_Valve,
                             RetractOutput => InternalOutput.bLowCV_Block1_Up_Valve);
cylinder.List.fbLowCV_Block1.IsDoubleValve := TRUE;

cylinder.List.fbLowCV_Block2(xDone =>,
                             xBusy =>,
                             xError =>CylinderStatus.LowCV_Block2.Error,
                             xEnable :=,
                             FrontSensor :=,
                             RearSensor := INPUT.bLowCV_Block2_RearSensor,
                             SetupPara := CurrentData.Cylinders.LowCV_Block2,
                             CurrentCylinderType =>,
                             InFrontPosition =>CylinderStatus.LowCV_Block2.InFrontPosition,
                             InRearPosition =>CylinderStatus.LowCV_Block2.InRearPosition,
                             ExtendOutput => InternalOutput.bLowCV_Block2_Down_Valve,
                             RetractOutput => InternalOutput.bLowCV_Block2_Up_Valve);
cylinder.List.fbLowCV_Block2.IsDoubleValve := TRUE;

cylinder.List.fbAllocateRobot_LeftVert1(xDone =>,
                                        xBusy =>,
                                        xError =>CylinderStatus.AllocateRobot_LeftVert1.Error,
                                        xEnable :=,
                                        FrontSensor := INPUT.bAllocateRobot_LeftVert1_LowSensor,
                                        RearSensor := INPUT.bAllocateRobot_LeftVert1_HighSensor,
                                        SetupPara := CurrentData.Cylinders.AllocateRobot_LeftVert1,
                                        CurrentCylinderType =>,
                                        InFrontPosition =>CylinderStatus.AllocateRobot_LeftVert1.InFrontPosition,
                                        InRearPosition =>CylinderStatus.AllocateRobot_LeftVert1.InRearPosition,
                                        ExtendOutput => InternalOutput.bAllocateRobot_LeftVert1_Valve,
                                        RetractOutput =>);

cylinder.List.fbAllocateRobot_LeftVert2(xDone =>,
                                        xBusy =>,
                                        xError =>CylinderStatus.AllocateRobot_LeftVert2.Error,
                                        xEnable :=,
                                        FrontSensor := input.bAllocateRobot_LeftVert2_LowSensor,
                                        RearSensor := input.bAllocateRobot_LeftVert2_HighSensor,
                                        SetupPara := CurrentData.Cylinders.AllocateRobot_LeftVert2,
                                        CurrentCylinderType =>,
                                        InFrontPosition =>CylinderStatus.AllocateRobot_LeftVert2.InFrontPosition,
                                        InRearPosition =>CylinderStatus.AllocateRobot_LeftVert2.InRearPosition,
                                        ExtendOutput => InternalOutput.bAllocateRobot_LeftVert2_Valve,
                                        RetractOutput =>);

cylinder.List.fbAllocateRobot_RightVert1(xDone =>,
                                         xBusy =>,
                                         xError =>CylinderStatus.AllocateRobot_RightVert1.Error,
                                         xEnable :=,
                                         FrontSensor := input.bAllocateRobot_RightVert1_LowSensor,
                                         RearSensor := input.bAllocateRobot_RightVert1_HighSensor,
                                         SetupPara := CurrentData.Cylinders.AllocateRobot_RightVert1,
                                         CurrentCylinderType =>,
                                         InFrontPosition =>CylinderStatus.AllocateRobot_RightVert1.InFrontPosition,
                                         InRearPosition =>CylinderStatus.AllocateRobot_RightVert1.InRearPosition,
                                         ExtendOutput => InternalOutput.bAllocateRobot_RightVert1_Valve,
                                         RetractOutput =>);

cylinder.List.fbAllocateRobot_RightVert2(xDone =>,
                                         xBusy =>,
                                         xError =>CylinderStatus.AllocateRobot_RightVert2.Error,
                                         xEnable :=,
                                         FrontSensor := input.bAllocateRobot_RightVert2_LowSensor,
                                         RearSensor := input.bAllocateRobot_RightVert2_HighSensor,
                                         SetupPara := CurrentData.Cylinders.AllocateRobot_RightVert2,
                                         CurrentCylinderType =>,
                                         InFrontPosition =>CylinderStatus.AllocateRobot_RightVert2.InFrontPosition,
                                         InRearPosition =>CylinderStatus.AllocateRobot_RightVert2.InRearPosition,
                                         ExtendOutput => InternalOutput.bAllocateRobot_RightVert2_Valve,
                                         RetractOutput =>);

cylinder.List.fbAllocateRobot_LeftClamp1(xDone =>,
                                         xBusy =>,
                                         xError =>CylinderStatus.AllocateRobot_LeftClamp1.Error,
                                         xEnable :=,
                                         FrontSensor :=,
                                         RearSensor :=,
                                         SetupPara := CurrentData.Cylinders.AllocateRobot_LeftClamp1,
                                         CurrentCylinderType =>,
                                         InFrontPosition =>CylinderStatus.AllocateRobot_LeftClamp1.InFrontPosition,
                                         InRearPosition =>CylinderStatus.AllocateRobot_LeftClamp1.InRearPosition,
                                         ExtendOutput => InternalOutput.bAllocateRobot_LeftClamp1_Close_Valve,
                                         RetractOutput => InternalOutput.bAllocateRobot_LeftClamp1_Open_Valve);
cylinder.List.fbAllocateRobot_LeftClamp1.IsDoubleValve := TRUE;

cylinder.List.fbAllocateRobot_LeftClamp2(xDone =>,
                                         xBusy =>,
                                         xError =>CylinderStatus.AllocateRobot_LeftClamp2.Error,
                                         xEnable :=,
                                         FrontSensor :=,
                                         RearSensor :=,
                                         SetupPara := CurrentData.Cylinders.AllocateRobot_LeftClamp2,
                                         CurrentCylinderType =>,
                                         InFrontPosition =>CylinderStatus.AllocateRobot_LeftClamp2.InFrontPosition,
                                         InRearPosition =>CylinderStatus.AllocateRobot_LeftClamp2.InRearPosition,
                                         ExtendOutput => InternalOutput.bAllocateRobot_LeftClamp2_Close_Valve,
                                         RetractOutput => InternalOutput.bAllocateRobot_LeftClamp2_Open_Valve);
cylinder.List.fbAllocateRobot_LeftClamp2.IsDoubleValve := TRUE;

cylinder.List.fbAllocateRobot_RightClamp1(xDone =>,
                                          xBusy =>,
                                          xError =>CylinderStatus.AllocateRobot_RightClamp1.Error,
                                          xEnable :=,
                                          FrontSensor :=,
                                          RearSensor :=,
                                          SetupPara := CurrentData.Cylinders.AllocateRobot_RightClamp1,
                                          CurrentCylinderType =>,
                                          InFrontPosition =>CylinderStatus.AllocateRobot_RightClamp1.InFrontPosition,
                                          InRearPosition =>CylinderStatus.AllocateRobot_RightClamp1.InRearPosition,
                                          ExtendOutput => InternalOutput.bAllocateRobot_RightClamp1_Close_Valve,
                                          RetractOutput => InternalOutput.bAllocateRobot_RightClamp1_Open_Valve);
cylinder.List.fbAllocateRobot_RightClamp1.IsDoubleValve := TRUE;

cylinder.List.fbAllocateRobot_RightClamp2(xDone =>,
                                          xBusy =>,
                                          xError =>CylinderStatus.AllocateRobot_RightClamp2.Error,
                                          xEnable :=,
                                          FrontSensor :=,
                                          RearSensor :=,
                                          SetupPara := CurrentData.Cylinders.AllocateRobot_RightClamp2,
                                          CurrentCylinderType =>,
                                          InFrontPosition =>CylinderStatus.AllocateRobot_RightClamp2.InFrontPosition,
                                          InRearPosition =>CylinderStatus.AllocateRobot_RightClamp2.InRearPosition,
                                          ExtendOutput => InternalOutput.bAllocateRobot_RightClamp2_Close_Valve,
                                          RetractOutput => InternalOutput.bAllocateRobot_RightClamp2_Open_Valve);
cylinder.List.fbAllocateRobot_RightClamp2.IsDoubleValve := TRUE;

cylinder.List.fbRoundBelt_WorkZone_Press(xDone =>,
                                         xBusy =>,
                                         xError =>CylinderStatus.RoundBelt_WorkZone_Press.Error,
                                         xEnable :=,
                                         FrontSensor :=,
                                         RearSensor := input.bRoundBelt_WorkZonePress_RearSensor,
                                         SetupPara := CurrentData.Cylinders.RoundBelt_WorkZone_Press,
                                         CurrentCylinderType =>,
                                         InFrontPosition =>CylinderStatus.RoundBelt_WorkZone_Press.InFrontPosition,
                                         InRearPosition =>CylinderStatus.RoundBelt_WorkZone_Press.InRearPosition,
                                         ExtendOutput => InternalOutput.bRoundBelt_WorkZone_Press_Valve,
                                         RetractOutput =>);

cylinder.List.fbRoundBelt_WorkZone_Plug(xDone =>,
                                        xBusy =>,
                                        xError =>CylinderStatus.RoundBelt_WorkZone_Plug.Error,
                                        xEnable :=,
                                        FrontSensor := input.bRoundBelt_WorkZonePlug_frontSensor,
                                        RearSensor := INPUT.bRoundBelt_WorkZonePlug_RearSensor,
                                        SetupPara := CurrentData.Cylinders.RoundBelt_WorkZone_Plug,
                                        CurrentCylinderType =>,
                                        InFrontPosition =>CylinderStatus.RoundBelt_WorkZone_Plug.InFrontPosition,
                                        InRearPosition =>CylinderStatus.RoundBelt_WorkZone_Plug.InRearPosition,
                                        ExtendOutput => InternalOutput.bRoundBelt_WorkZone_Plug_Valve,
                                        RetractOutput =>);

cylinder.List.fbRoundBelt_ChargeZone_Plug(xDone =>,
                                          xBusy =>,
                                          xError =>CylinderStatus.RoundBelt_ChargeZone_Plug.Error,
                                          xEnable :=,
                                          FrontSensor := INPUT.bRoundBelt_ChangeZonePlug_FrontSensor,
                                          RearSensor := input.bRoundBelt_ChangeZonePlug_RearSensor,
                                          SetupPara := CurrentData.Cylinders.RoundBelt_ChargeZone_Plug,
                                          CurrentCylinderType =>,
                                          InFrontPosition =>CylinderStatus.RoundBelt_ChargeZone_Plug.InFrontPosition,
                                          InRearPosition =>CylinderStatus.RoundBelt_ChargeZone_Plug.InRearPosition,
                                          ExtendOutput => InternalOutput.bRoundBelt_ChargeZone_Plug_Valve,
                                          RetractOutput =>);

cylinder.List.fbRoundBelt_TransmitCVZone_Plug(xDone =>,
                                              xBusy =>,
                                              xError =>CylinderStatus.RoundBelt_TransmitCVZone_Plug.Error,
                                              xEnable :=,
                                              FrontSensor := input.bRoundBelt_TransmitCVZonePlug_FrontSensor,
                                              RearSensor := INPUT.bRoundBelt_TransmitCVZonePlug_RearSensor,
                                              SetupPara := CurrentData.Cylinders.RoundBelt_TransmitCVZone_Plug,
                                              CurrentCylinderType =>,
                                              InFrontPosition =>CylinderStatus.RoundBelt_TransmitCVZone_Plug.InFrontPosition,
                                              InRearPosition =>CylinderStatus.RoundBelt_TransmitCVZone_Plug.InRearPosition,
                                              ExtendOutput => InternalOutput.bRoundBelt_TransmitCVZone_Plug_Valve,
                                              RetractOutput =>);

cylinder.List.fbOutRobot_AsideVert(xDone =>,
                                   xBusy =>,
                                   xError =>CylinderStatus.OutRobot_AsideVert.Error,
                                   xEnable :=,
                                   FrontSensor := INPUT.bOutRobot_AsideVert_LowSensor,
                                   RearSensor := input.bOutRobot_AsideVert_highSensor,
                                   SetupPara := CurrentData.Cylinders.OutRobot_AsideVert,
                                   CurrentCylinderType =>,
                                   InFrontPosition =>CylinderStatus.OutRobot_AsideVert.InFrontPosition,
                                   InRearPosition =>CylinderStatus.OutRobot_AsideVert.InRearPosition,
                                   ExtendOutput => InternalOutput.bOutRobot_AsideVert_Valve,
                                   RetractOutput =>);

cylinder.List.fbOutRobot_BsideVert(xDone =>,
                                   xBusy =>,
                                   xError =>CylinderStatus.OutRobot_BsideVert.Error,
                                   xEnable :=,
                                   FrontSensor := input.bOutRobot_BsideVert_LowSensor,
                                   RearSensor := INPUT.bOutRobot_BsideVert_HighSensor,
                                   SetupPara := CurrentData.Cylinders.OutRobot_BsideVert,
                                   CurrentCylinderType =>,
                                   InFrontPosition =>CylinderStatus.OutRobot_BsideVert.InFrontPosition,
                                   InRearPosition =>CylinderStatus.OutRobot_BsideVert.InRearPosition,
                                   ExtendOutput => InternalOutput.bOutRobot_BsideVert_Valve,
                                   RetractOutput =>);

cylinder.List.fbOutRobot_AsideClamp(xDone =>,
                                    xBusy =>,
                                    xError =>CylinderStatus.OutRobot_AsideClamp.Error,
                                    xEnable :=,
                                    FrontSensor :=,
                                    RearSensor := input.bOutRobot_AsideClamp_RearSensor,
                                    SetupPara := CurrentData.Cylinders.OutRobot_AsideClamp,
                                    CurrentCylinderType =>,
                                    InFrontPosition =>CylinderStatus.OutRobot_AsideClamp.InFrontPosition,
                                    InRearPosition =>CylinderStatus.OutRobot_AsideClamp.InRearPosition,
                                    ExtendOutput => InternalOutput.bOutRobot_AsideClamp_Close_Valve,
                                    RetractOutput => InternalOutput.bOutRobot_AsideClamp_Open_Valve);
cylinder.List.fbOutRobot_AsideClamp.IsDoubleValve := TRUE;

cylinder.List.fbOutRobot_BsideClamp(xDone =>,
                                    xBusy =>,
                                    xError =>CylinderStatus.OutRobot_BsideClamp.Error,
                                    xEnable :=,
                                    FrontSensor :=,
                                    RearSensor := input.bOutRobot_BsideClamp_RearSensor,
                                    SetupPara := CurrentData.Cylinders.OutRobot_BsideClamp,
                                    CurrentCylinderType =>,
                                    InFrontPosition =>CylinderStatus.OutRobot_BsideClamp.InFrontPosition,
                                    InRearPosition =>CylinderStatus.OutRobot_BsideClamp.InRearPosition,
                                    ExtendOutput => InternalOutput.bOutRobot_BsideClamp_Close_Valve,
                                    RetractOutput => InternalOutput.bOutRobot_BsideClamp_Open_Valve);
cylinder.List.fbOutRobot_BsideClamp.IsDoubleValve := TRUE;

cylinder.List.fbTransmitCV_CamaraHoriz(xDone =>,
                                       xBusy =>,
                                       xError =>CylinderStatus.TransmitCV_CamaraHoriz.Error,
                                       xEnable :=,
                                       FrontSensor :=input.bTransmit_CamaraHorizDifferentSizeSide_Sensor,
                                       RearSensor := input.bTransmit_CamaraHorizSameSizeSide_Sensor,
                                       SetupPara := CurrentData.Cylinders.TransmitCV_CamaraHoriz,
                                       CurrentCylinderType =>,
                                       InFrontPosition =>CylinderStatus.TransmitCV_CamaraHoriz.InFrontPosition,
                                       InRearPosition =>CylinderStatus.TransmitCV_CamaraHoriz.InRearPosition,
                                       ExtendOutput => InternalOutput.bTransmitCV_CamaraHorizDifferentSide_Valve,
                                       RetractOutput => InternalOutput.bTransmitCV_CamaraHorizSameSizeSide_Valve);
cylinder.List.fbTransmitCV_CamaraHoriz.IsDoubleValve := TRUE;

cylinder.List.fbDifferentSizeCV_Press2(xDone =>,
                                       xBusy =>,
                                       xError =>CylinderStatus.DifferentSizeCV_Press2.Error,
                                       xEnable :=,
                                       FrontSensor :=,
                                       RearSensor :=,
                                       SetupPara := CurrentData.Cylinders.DifferentSizeCV_Press2,
                                       CurrentCylinderType =>,
                                       InFrontPosition =>CylinderStatus.DifferentSizeCV_Press2.InFrontPosition,
                                       InRearPosition =>CylinderStatus.DifferentSizeCV_Press2.InRearPosition,
                                       ExtendOutput => InternalOutput.bDifferentSizeCV_Press2_Valve,
                                       RetractOutput =>);

cylinder.List.fbDifferentSizeCV_Press1(xDone =>,
                                       xBusy =>,
                                       xError =>CylinderStatus.DifferentSizeCV_Press1.Error,
                                       xEnable :=,
                                       FrontSensor :=,
                                       RearSensor :=,
                                       SetupPara := CurrentData.Cylinders.DifferentSizeCV_Press1,
                                       CurrentCylinderType =>,
                                       InFrontPosition =>CylinderStatus.DifferentSizeCV_Press1.InFrontPosition,
                                       InRearPosition =>CylinderStatus.DifferentSizeCV_Press1.InRearPosition,
                                       ExtendOutput => InternalOutput.bDifferentSizeCV_Press1_Valve,
                                       RetractOutput =>);

cylinder.List.fbDifferentSizeCV_Block1(xDone =>,
                                       xBusy =>,
                                       xError =>CylinderStatus.DifferentSizeCV_Block1.Error,
                                       xEnable :=,
                                       FrontSensor :=,
                                       RearSensor := INPUT.bDifferentCV_Block_RearSensor,
                                       SetupPara := CurrentData.Cylinders.DifferentSizeCV_Block1,
                                       CurrentCylinderType =>,
                                       InFrontPosition =>CylinderStatus.DifferentSizeCV_Block1.InFrontPosition,
                                       InRearPosition =>CylinderStatus.DifferentSizeCV_Block1.InRearPosition,
                                       ExtendOutput => InternalOutput.bDifferentSizeCV_Block1_Valve,
                                       RetractOutput =>);

cylinder.List.fbSameSizeCV_Press4(xDone =>,
                                  xBusy =>,
                                  xError =>CylinderStatus.SameSizeCV_Press4.Error,
                                  xEnable :=,
                                  FrontSensor :=,
                                  RearSensor :=,
                                  SetupPara := CurrentData.Cylinders.SameSizeCV_Press4,
                                  CurrentCylinderType =>,
                                  InFrontPosition =>CylinderStatus.SameSizeCV_Press4.InFrontPosition,
                                  InRearPosition =>CylinderStatus.SameSizeCV_Press4.InRearPosition,
                                  ExtendOutput => InternalOutput.bSameSizeCV_Press4_Valve,
                                  RetractOutput =>);

cylinder.List.fbSameSizeCV_Press3(xDone =>,
                                  xBusy =>,
                                  xError =>CylinderStatus.SameSizeCV_Press3.Error,
                                  xEnable :=,
                                  FrontSensor :=,
                                  RearSensor :=,
                                  SetupPara := CurrentData.Cylinders.SameSizeCV_Press3,
                                  CurrentCylinderType =>,
                                  InFrontPosition =>CylinderStatus.SameSizeCV_Press3.InFrontPosition,
                                  InRearPosition =>CylinderStatus.SameSizeCV_Press3.InRearPosition,
                                  ExtendOutput => InternalOutput.bSameSizeCV_Press3_Valve,
                                  RetractOutput =>);

cylinder.List.fbSameSizeCV_Press2(xDone =>,
                                  xBusy =>,
                                  xError =>CylinderStatus.SameSizeCV_Press2.Error,
                                  xEnable :=,
                                  FrontSensor :=,
                                  RearSensor :=,
                                  SetupPara := CurrentData.Cylinders.SameSizeCV_Press2,
                                  CurrentCylinderType =>,
                                  InFrontPosition =>CylinderStatus.SameSizeCV_Press2.InFrontPosition,
                                  InRearPosition =>CylinderStatus.SameSizeCV_Press2.InRearPosition,
                                  ExtendOutput => InternalOutput.bSameSizeCV_Press2_Valve,
                                  RetractOutput =>);

cylinder.List.fbSameSizeCV_Press1(xDone =>,
                                  xBusy =>,
                                  xError =>CylinderStatus.SameSizeCV_Press1.Error,
                                  xEnable :=,
                                  FrontSensor :=,
                                  RearSensor :=,
                                  SetupPara := CurrentData.Cylinders.SameSizeCV_Press1,
                                  CurrentCylinderType =>,
                                  InFrontPosition =>CylinderStatus.SameSizeCV_Press1.InFrontPosition,
                                  InRearPosition =>CylinderStatus.SameSizeCV_Press1.InRearPosition,
                                  ExtendOutput => InternalOutput.bSameSizeCV_Press1_Valve,
                                  RetractOutput =>);

cylinder.List.fbSameSizeCV_Block2(xDone =>,
                                  xBusy =>,
                                  xError =>CylinderStatus.SameSizeCV_Block2.Error,
                                  xEnable :=,
                                  FrontSensor :=,
                                  RearSensor := input.bSameSizeCVBlock2_RearSensor,
                                  SetupPara := CurrentData.Cylinders.SameSizeCV_Block2,
                                  CurrentCylinderType =>,
                                  InFrontPosition =>CylinderStatus.SameSizeCV_Block2.InFrontPosition,
                                  InRearPosition =>CylinderStatus.SameSizeCV_Block2.InRearPosition,
                                  ExtendOutput => InternalOutput.bSameSizeCV_Block2_Valve,
                                  RetractOutput =>);

cylinder.List.fbSameSizeCV_Block1(xDone =>,
                                  xBusy =>,
                                  xError =>CylinderStatus.SameSizeCV_Block1.Error,
                                  xEnable :=,
                                  FrontSensor :=,
                                  RearSensor := input.bSameSizeCVBlock1_RearSensor,
                                  SetupPara := CurrentData.Cylinders.SameSizeCV_Block1,
                                  CurrentCylinderType =>,
                                  InFrontPosition =>CylinderStatus.SameSizeCV_Block1.InFrontPosition,
                                  InRearPosition =>CylinderStatus.SameSizeCV_Block1.InRearPosition,
                                  ExtendOutput => InternalOutput.bSameSizeCV_Block1_Valve,
                                  RetractOutput =>);

cylinder.List.fbTurntable_Press(xDone =>,
                                xBusy =>,
                                xError =>CylinderStatus.Turntable_Press.Error,
                                xEnable :=,
                                FrontSensor :=,
                                RearSensor := input.bTurnTable_Press_RearSensor,
                                SetupPara := CurrentData.Cylinders.Turntable_Press,
                                CurrentCylinderType =>,
                                InFrontPosition =>CylinderStatus.Turntable_Press.InFrontPosition,
                                InRearPosition =>CylinderStatus.Turntable_Press.InRearPosition,
                                ExtendOutput => InternalOutput.bTurntable_Press_Valve,
                                RetractOutput =>);
END_ACTION

ACTION A02_Motor:
Motor.List.WareHouseCV_10(xDone =>,
                          xBusy =>,
                          xError => MotorStatus.WareHouseCV_10.Error,
                          xEnable :=,
                          OverLoadSignal :=,
                          SetupPara :=,
                          InForWard =>MotorStatus.WareHouseCV_10.InForward,
                          InBackWard =>MotorStatus.WareHouseCV_10.InBackward,
                          InStopped =>MotorStatus.WareHouseCV_10.InStopped,
                          ForWardOutput => InternalOutput.bWareHouseCV10_Fwd,
                          BackWardOutput => InternalOutput.bWareHouseCV10_Rev);

Motor.List.WareHouseCV_09(xDone =>,
                          xBusy =>,
                          xError =>MotorStatus.WareHouseCV_09.Error,
                          xEnable :=,
                          OverLoadSignal :=,
                          SetupPara :=,
                          InForWard =>MotorStatus.WareHouseCV_09.InForward,
                          InBackWard =>MotorStatus.WareHouseCV_09.InBackward,
                          InStopped =>MotorStatus.WareHouseCV_09.InStopped,
                          ForWardOutput =>InternalOutput.bWareHouseCV9_Fwd,
                          BackWardOutput =>InternalOutput.bWareHouseCV9_Rev);

Motor.List.WareHouseCV_08(xDone =>,
                          xBusy =>,
                          xError =>MotorStatus.WareHouseCV_08.Error,
                          xEnable :=,
                          OverLoadSignal :=,
                          SetupPara :=,
                          InForWard =>MotorStatus.WareHouseCV_08.InForward,
                          InBackWard =>MotorStatus.WareHouseCV_08.InBackward,
                          InStopped =>MotorStatus.WareHouseCV_08.InStopped,
                          ForWardOutput =>InternalOutput.bWareHouseCV8_Fwd,
                          BackWardOutput =>InternalOutput.bWareHouseCV8_Rev);

Motor.List.WareHouseCV_07(xDone =>,
                          xBusy =>,
                          xError =>MotorStatus.WareHouseCV_07.Error,
                          xEnable :=,
                          OverLoadSignal :=,
                          SetupPara :=,
                          InForWard =>MotorStatus.WareHouseCV_07.InForward,
                          InBackWard =>MotorStatus.WareHouseCV_07.InBackward,
                          InStopped =>MotorStatus.WareHouseCV_07.InStopped,
                          ForWardOutput =>InternalOutput.bWareHouseCV7_Fwd,
                          BackWardOutput =>InternalOutput.bWareHouseCV7_Rev);

Motor.List.WareHouseCV_06(xDone =>,
                          xBusy =>,
                          xError =>MotorStatus.WareHouseCV_06.Error,
                          xEnable :=,
                          OverLoadSignal :=,
                          SetupPara :=,
                          InForWard =>MotorStatus.WareHouseCV_06.InForward,
                          InBackWard =>MotorStatus.WareHouseCV_06.InBackward,
                          InStopped =>MotorStatus.WareHouseCV_06.InStopped,
                          ForWardOutput =>InternalOutput.bWareHouseCV6_Fwd,
                          BackWardOutput =>InternalOutput.bWareHouseCV6_Rev);

Motor.List.WareHouseCV_05(xDone =>,
                          xBusy =>,
                          xError =>MotorStatus.WareHouseCV_05.Error,
                          xEnable :=,
                          OverLoadSignal :=,
                          SetupPara :=,
                          InForWard =>MotorStatus.WareHouseCV_05.InForward,
                          InBackWard =>MotorStatus.WareHouseCV_05.InBackward,
                          InStopped =>MotorStatus.WareHouseCV_05.InStopped,
                          ForWardOutput =>InternalOutput.bWareHouseCV5_Fwd,
                          BackWardOutput =>InternalOutput.bWareHouseCV5_Rev);

Motor.List.WareHouseCV_04(xDone =>,
                          xBusy =>,
                          xError =>MotorStatus.WareHouseCV_04.Error,
                          xEnable :=,
                          OverLoadSignal :=,
                          SetupPara :=,
                          InForWard =>MotorStatus.WareHouseCV_04.InForward,
                          InBackWard =>MotorStatus.WareHouseCV_04.InBackward,
                          InStopped =>MotorStatus.WareHouseCV_04.InStopped,
                          ForWardOutput =>InternalOutput.bWareHouseCV4_Fwd,
                          BackWardOutput =>InternalOutput.bWareHouseCV4_Rev);

Motor.List.WareHouseCV_03(xDone =>,
                          xBusy =>,
                          xError =>MotorStatus.WareHouseCV_03.Error,
                          xEnable :=,
                          OverLoadSignal :=,
                          SetupPara :=,
                          InForWard =>MotorStatus.WareHouseCV_03.InForward,
                          InBackWard =>MotorStatus.WareHouseCV_03.InBackward,
                          InStopped =>MotorStatus.WareHouseCV_03.InStopped,
                          ForWardOutput =>InternalOutput.bWareHouseCV3_Fwd,
                          BackWardOutput =>InternalOutput.bWareHouseCV3_Rev);

Motor.List.WareHouseCV_02(xDone =>,
                          xBusy =>,
                          xError =>MotorStatus.WareHouseCV_02.Error,
                          xEnable :=,
                          OverLoadSignal :=,
                          SetupPara :=,
                          InForWard =>MotorStatus.WareHouseCV_02.InForward,
                          InBackWard =>MotorStatus.WareHouseCV_02.InBackward,
                          InStopped =>MotorStatus.WareHouseCV_02.InStopped,
                          ForWardOutput =>InternalOutput.bWareHouseCV2_Fwd,
                          BackWardOutput =>InternalOutput.bWareHouseCV2_Rev);

Motor.List.WareHouseCV_01(xDone =>,
                          xBusy =>,
                          xError =>MotorStatus.WareHouseCV_01.Error,
                          xEnable :=,
                          OverLoadSignal :=,
                          SetupPara :=,
                          InForWard =>MotorStatus.WareHouseCV_01.InForward,
                          InBackWard =>MotorStatus.WareHouseCV_01.InBackward,
                          InStopped =>MotorStatus.WareHouseCV_01.InStopped,
                          ForWardOutput =>InternalOutput.bWareHouseCV1_Fwd,
                          BackWardOutput =>InternalOutput.bWareHouseCV1_Rev);

Motor.List.WareHouseCV_20(xDone =>,
                          xBusy =>,
                          xError =>MotorStatus.WareHouseCV_20.Error,
                          xEnable :=,
                          OverLoadSignal :=,
                          SetupPara :=,
                          InForWard =>MotorStatus.WareHouseCV_20.InForward,
                          InBackWard =>MotorStatus.WareHouseCV_20.InBackward,
                          InStopped =>MotorStatus.WareHouseCV_20.InStopped,
                          ForWardOutput =>InternalOutput.bWareHouseCV20_Fwd,
                          BackWardOutput =>InternalOutput.bWareHouseCV20_Rev);

Motor.List.WareHouseCV_19(xDone =>,
                          xBusy =>,
                          xError =>MotorStatus.WareHouseCV_19.Error,
                          xEnable :=,
                          OverLoadSignal :=,
                          SetupPara :=,
                          InForWard =>MotorStatus.WareHouseCV_19.InForward,
                          InBackWard =>MotorStatus.WareHouseCV_19.InBackward,
                          InStopped =>MotorStatus.WareHouseCV_19.InStopped,
                          ForWardOutput =>InternalOutput.bWareHouseCV19_Fwd,
                          BackWardOutput =>InternalOutput.bWareHouseCV19_Rev);

Motor.List.WareHouseCV_18(xDone =>,
                          xBusy =>,
                          xError =>MotorStatus.WareHouseCV_18.Error,
                          xEnable :=,
                          OverLoadSignal :=,
                          SetupPara :=,
                          InForWard =>MotorStatus.WareHouseCV_18.InForward,
                          InBackWard =>MotorStatus.WareHouseCV_18.InBackward,
                          InStopped =>MotorStatus.WareHouseCV_18.InStopped,
                          ForWardOutput =>InternalOutput.bWareHouseCV18_Fwd,
                          BackWardOutput =>InternalOutput.bWareHouseCV18_Rev);

Motor.List.WareHouseCV_17(xDone =>,
                          xBusy =>,
                          xError =>MotorStatus.WareHouseCV_17.Error,
                          xEnable :=,
                          OverLoadSignal :=,
                          SetupPara :=,
                          InForWard =>MotorStatus.WareHouseCV_17.InForward,
                          InBackWard =>MotorStatus.WareHouseCV_17.InBackward,
                          InStopped =>MotorStatus.WareHouseCV_17.InStopped,
                          ForWardOutput =>InternalOutput.bWareHouseCV17_Fwd,
                          BackWardOutput =>InternalOutput.bWareHouseCV17_Rev);

Motor.List.WareHouseCV_16(xDone =>,
                          xBusy =>,
                          xError =>MotorStatus.WareHouseCV_16.Error,
                          xEnable :=,
                          OverLoadSignal :=,
                          SetupPara :=,
                          InForWard =>MotorStatus.WareHouseCV_16.InForward,
                          InBackWard =>MotorStatus.WareHouseCV_16.InBackward,
                          InStopped =>MotorStatus.WareHouseCV_16.InStopped,
                          ForWardOutput =>InternalOutput.bWareHouseCV16_Fwd,
                          BackWardOutput =>InternalOutput.bWareHouseCV16_Rev);

Motor.List.WareHouseCV_15(xDone =>,
                          xBusy =>,
                          xError =>MotorStatus.WareHouseCV_15.Error,
                          xEnable :=,
                          OverLoadSignal :=,
                          SetupPara :=,
                          InForWard =>MotorStatus.WareHouseCV_15.InForward,
                          InBackWard =>MotorStatus.WareHouseCV_15.InBackward,
                          InStopped =>MotorStatus.WareHouseCV_15.InStopped,
                          ForWardOutput =>InternalOutput.bWareHouseCV15_Fwd,
                          BackWardOutput =>InternalOutput.bWareHouseCV15_Rev);

Motor.List.WareHouseCV_14(xDone =>,
                          xBusy =>,
                          xError =>MotorStatus.WareHouseCV_14.Error,
                          xEnable :=,
                          OverLoadSignal :=,
                          SetupPara :=,
                          InForWard =>MotorStatus.WareHouseCV_14.InForward,
                          InBackWard =>MotorStatus.WareHouseCV_14.InBackward,
                          InStopped =>MotorStatus.WareHouseCV_14.InStopped,
                          ForWardOutput =>InternalOutput.bWareHouseCV14_Fwd,
                          BackWardOutput =>InternalOutput.bWareHouseCV14_Rev);

Motor.List.WareHouseCV_13(xDone =>,
                          xBusy =>,
                          xError =>MotorStatus.WareHouseCV_13.Error,
                          xEnable :=,
                          OverLoadSignal :=,
                          SetupPara :=,
                          InForWard =>MotorStatus.WareHouseCV_13.InForward,
                          InBackWard =>MotorStatus.WareHouseCV_13.InBackward,
                          InStopped =>MotorStatus.WareHouseCV_13.InStopped,
                          ForWardOutput =>InternalOutput.bWareHouseCV13_Fwd,
                          BackWardOutput =>InternalOutput.bWareHouseCV13_Rev);

Motor.List.WareHouseCV_12(xDone =>,
                          xBusy =>,
                          xError =>MotorStatus.WareHouseCV_12.Error,
                          xEnable :=,
                          OverLoadSignal :=,
                          SetupPara :=,
                          InForWard =>MotorStatus.WareHouseCV_12.InForward,
                          InBackWard =>MotorStatus.WareHouseCV_12.InBackward,
                          InStopped =>MotorStatus.WareHouseCV_12.InStopped,
                          ForWardOutput =>InternalOutput.bWareHouseCV12_Fwd,
                          BackWardOutput =>InternalOutput.bWareHouseCV12_Rev);

Motor.List.WareHouseCV_11(xDone =>,
                          xBusy =>,
                          xError =>MotorStatus.WareHouseCV_11.Error,
                          xEnable :=,
                          OverLoadSignal :=,
                          SetupPara :=,
                          InForWard =>MotorStatus.WareHouseCV_11.InForward,
                          InBackWard =>MotorStatus.WareHouseCV_11.InBackward,
                          InStopped =>MotorStatus.WareHouseCV_11.InStopped,
                          ForWardOutput =>InternalOutput.bWareHouseCV11_Fwd,
                          BackWardOutput =>InternalOutput.bWareHouseCV11_Rev);

Motor.List.UpCV(xDone =>,
                xBusy =>,
                xError =>MotorStatus.UpCV.Error,
                xEnable :=,
                OverLoadSignal :=,
                SetupPara :=,
                InForWard =>MotorStatus.UpCV.InForward,
                InBackWard =>MotorStatus.UpCV.InBackward,
                InStopped =>MotorStatus.UpCV.InStopped,
                ForWardOutput =>InternalOutput.bUpCV_Fwd,
                BackWardOutput =>InternalOutput.bUpCV_Rev);

Motor.List.LowCV(xDone =>,
                xBusy =>,
                xError =>MotorStatus.LowCV.Error,
                xEnable :=,
                OverLoadSignal :=,
                SetupPara :=,
                InForWard =>MotorStatus.LowCV.InForward,
                InBackWard =>MotorStatus.LowCV.InBackward,
                InStopped =>MotorStatus.LowCV.InStopped,
                ForWardOutput =>InternalOutput.bLowCV_Fwd,
                BackWardOutput =>InternalOutput.bLowCV_Rev);

Motor.List.PullOutCV_A(xDone =>,
						xBusy =>,
						xError =>MotorStatus.PullOutCV_A.Error,
						xEnable :=,
						OverLoadSignal :=,
						SetupPara :=,
						InForWard =>MotorStatus.PullOutCV_A.InForward,
						InBackWard =>MotorStatus.PullOutCV_A.InBackward,
						InStopped =>MotorStatus.PullOutCV_A.InStopped,
						ForWardOutput =>InternalOutput.bPullOutCV_A_Fwd,
						BackWardOutput =>InternalOutput.bPullOutCV_A_Rev);

Motor.List.PullOutCV_B(xDone =>,
						xBusy =>,
						xError =>MotorStatus.PullOutCV_B.Error,
						xEnable :=,
						OverLoadSignal :=,
						SetupPara :=,
						InForWard =>MotorStatus.PullOutCV_B.InForward,
						InBackWard =>MotorStatus.PullOutCV_B.InBackward,
						InStopped =>MotorStatus.PullOutCV_B.InStopped,
						ForWardOutput =>InternalOutput.bPullOutCV_B_Fwd,
						BackWardOutput =>InternalOutput.bPullOutCV_B_Rev);

Motor.List.TransmitSameSideCV(xDone =>,
								xBusy =>,
								xError =>MotorStatus.TransmitSameSideCV.Error,
								xEnable :=,
								OverLoadSignal :=,
								SetupPara :=,
								InForWard =>MotorStatus.TransmitSameSideCV.InForward,
								InBackWard =>MotorStatus.TransmitSameSideCV.InBackward,
								InStopped =>MotorStatus.TransmitSameSideCV.InStopped,
								ForWardOutput =>InternalOutput.bTransmitCV_SameSizeSide_Fwd,
								BackWardOutput =>InternalOutput.bTransmitCV_SameSide_Rev);

Motor.List.TransmitDifferentSideCV(xDone =>,
									xBusy =>,
									xError =>MotorStatus.TransmitDifferentSideCV.Error,
									xEnable :=,
									OverLoadSignal :=,
									SetupPara :=,
									InForWard =>MotorStatus.TransmitDifferentSideCV.InForward,
									InBackWard =>MotorStatus.TransmitDifferentSideCV.InBackward,
									InStopped =>MotorStatus.TransmitDifferentSideCV.InStopped,
									ForWardOutput =>InternalOutput.bTransmitCV_DifferentSide_Fwd,
									BackWardOutput =>InternalOutput.bTransmitCV_DifferentSide_Rev);
END_ACTION

ACTION A03_FanucRobot:
FanucRobot.List.StorageRobot(
	Estop:= Machine_Estop (*OR Input.bStorage_EstopPb*), 
	OpMode:= , 
	Start:= Machine_Start , 
//	Reset:= Machine_Reset OR fbStorageArea.RobotResetCMD, 
//	Hold:= Machine_Stop, 
	Reset:= Machine_Reset OR fbStorageArea.RobotResetCMD OR tofResetDelay.Q, //Postpone reset signal to fanuc robot		
	Hold:=   NOT FanucRobot.List.StorageRobot.Error AND_THEN Machine_Stop, 		//Transport form Kinsus version to taixin
	ManualCtrl :=  GVL_HMI.Storage.Manual.FanucRobot,
	qEnable=> , 
	qFault=> ,

	E_Stop_Output=> StorageRobot_EStop, 
	Halt=> , 
	Error=> , 
	ErrorID=> );

FanucRobot.List.ShippingRobot(
	Estop:= Machine_Estop (*OR Input.bStorage_EstopPb*), 
	OpMode:= , 
	Start:= Machine_Start, 
	Reset:= Machine_Reset OR fbShippingArea.RobotResetCMD OR tofResetDelay.Q, 			//
	Hold:= NOT fanucrobot.List.ShippingRobot.Error AND_THEN Machine_Stop,
	ManualCtrl:= GVL_HMI.Shipping.Manual.FanucRobot, 
	qEnable=> , 
	qFault=> , 
	E_Stop_Output=> ShippingRobot_EStop, 
	Halt=> , 
	Error=> , 
	ErrorID=> );
END_ACTION

ACTION A04_OpPannel:
// E-Stop 
Machine_Estop := (NOT INPUT.bAllocate_EStopPb OR
                 NOT INPUT.bStorage_EstopPb OR
                 StorageRobot_EStop OR
                 ShippingRobot_EStop OR
                 GVL_ADS.OpPannel_Ctrl.EStopBtnStatus OR 
				NOT INPUT.bStorage_AirPressure_Ready) AND
                 NOT EnableSimulation;

// Stop
bSafetyDoorOpen := (NOT INPUT.bSafetyDoor1 OR
                   NOT INPUT.bSafetyDoor2 OR
                   NOT INPUT.bSafetyDoor3 OR
                   NOT INPUT.bSafetyDoor4 OR		
                   NOT INPUT.bSafetyDoor5 OR
                   NOT INPUT.bSafetyDoor6 OR
                   NOT INPUT.bSafetyDoor7 OR
                   NOT INPUT.bSafetyDoor8 OR
                   not INPUT.bSafetyDoor9 OR
                   not INPUT.bSafetyDoor10 OR
                   not INPUT.bSafetyDoor11 OR
                   not INPUT.bSafetyDoor12 OR
                   not INPUT.bSafetyDoor13 OR
                   not INPUT.bSafetyDoor14 OR
                   NOT INPUT.bAllocate_Electrical_Cabinet_SafetyDoor OR
                   NOT INPUT.bShippingRobot_ElectricalCabinet_SafetyDoor) AND
				   (NOT    GVL_HMI.Setup.Mechanical.stSafetyByPass.SafeDoorByPass)	;		//use Safedoor bypass

IF StopEdgeDetect.xRisingEdge THEN
    bStopMem := TRUE;
ELSIF ResetEdgeDetect.xRisingEdge THEN
    bStopMem := FALSE;
END_IF

Machine_Stop := INPUT.bAllocate_StopPb OR
                INPUT.bStorage_StopPb OR
                bSafetyDoorOpen OR
                xError OR
                GVL_ADS.OpPannel_Ctrl.StopBtnStatus;

// Reset
Machine_Reset :=
    INPUT.bAllocate_ResetPb OR INPUT.bStorage_ResetPb OR GVL_ADS.OpPannel_Ctrl.ResetBtnStatus;

// Start
Machine_Start :=
    INPUT.bAllocate_StartPb OR INPUT.bStorage_StartPb OR GVL_ADS.OpPannel_Ctrl.StartBtnStatus;

//IF xError THEN
//    InternalOutput.bAllocated_SignalTower_RedLamp := fbBlink_05.OUT;
//    InternalOutput.bStorage_SingleTower_RedLamp := fbBlink_05.OUT;
//	InternalOutput.bAllocated_StopPbLamp := fbBlink_05.OUT;
//	InternalOutput.bStorage_StopPbLamp := fbBlink_05.OUT;
//ELSIF bStopMem AND NOT xError THEN
//    InternalOutput.bAllocated_SignalTower_RedLamp := TRUE;
//    InternalOutput.bStorage_SingleTower_RedLamp := TRUE;
//	InternalOutput.bAllocated_StopPbLamp := TRUE;
//	InternalOutput.bStorage_StopPbLamp := TRUE;
//ELSE
//    InternalOutput.bAllocated_SignalTower_RedLamp := FALSE;
//    InternalOutput.bStorage_SingleTower_RedLamp := FALSE;
//	InternalOutput.bAllocated_StopPbLamp := FALSE;
//	InternalOutput.bStorage_StopPbLamp := FALSE;

//END_IF

InternalOutput.bAllocated_SignalTower_RedLamp := _RedLamp;
InternalOutput.bAllocated_SignalTower_YellowLamp := _YellowLamp;
InternalOutput.bAllocated_SignalTower_GreenLamp := _GreenLamp;
InternalOutput.bAllocated_Buzzer := _Buzz;
InternalOutput.bStorage_Buzzer := _Buzz;
InternalOutput.bStorage_SingleTower_RedLamp := _RedLamp;
InternalOutput.bStorage_SingleTower_YellowLamp := _YellowLamp;
InternalOutput.bStorage_SingleTower_GreenLamp := _GreenLamp;

InternalOutput.bAllocated_StopPbLamp := _RedLamp;
InternalOutput.bAllocated_StartPbLamp := _GreenLamp;
InternalOutput.bAllocated_ResetPbLamp := _YellowLamp;

InternalOutput.bStorage_ResetPbLamp := _YellowLamp;
InternalOutput.bStorage_StartPbLamp := _GreenLamp;
InternalOutput.bStorage_StopPbLamp := _RedLamp;

//postpone btn signal to Host
tofResetDelay.IN:=Machine_Reset;
tofStopDelay.IN :=Machine_Stop; 
tofStartDelay.IN:=Machine_Start;
tofResetDelay(PT:=T#3.2S);	
tofStopDelay(PT:=T#1S);	
tofStartDelay(PT:=T#1S);

GVL_ADS.OpPannel_Status.EStopBtnStatus := Machine_Estop;
GVL_ADS.OpPannel_Status.ResetBtnStatus := tofResetDelay.Q;
GVL_ADS.OpPannel_Status.StartBtnStatus := tofStartDelay.Q;
GVL_ADS.OpPannel_Status.StopBtnStatus  := tofStopDelay.Q;


fb_AllocateSignalTower(
	Enable:= , 
	LampRed:= _RedLamp, 
	LampYellow:= _YellowLamp, 
	LampGreen:= _GreenLamp, 
	Buzz:= _Buzz, 
	ForceCloseBuzz:= , 
	BuzzSwitchOnTime:= 5, 
	Vaild=> , 
	Error=> , 
	ErrorID=> );
END_ACTION

ACTION A05_Light:
//  Light 
InternalOutput.bStorage_EleBoxLight := GVL_HMI.Setup.Light.Storage_EleBoxLight_Off;
InternalOutput.bStorage_AreaLight := GVL_HMI.Setup.Light.Storage_AreaLight_Off;
InternalOutput.bAllocated_AreaLight := GVL_HMI.Setup.Light.Allocated_AreaLight_Off;

// Upcv CameraBlow
InternalOutput.bCamara_Blow := GVL_HMI.Storage.Manual.UpCV.CameraBlow;
END_ACTION

ACTION A10_ErrorHandler:
IF NOT ErrorTableInitDone THEN
	ErrorTableInitDone := M_General_AlarmRegister();
END_IF
M_General_AlarmRegister();
//Machine_Estop := ( NOT INPUT.bAllocate_EStopPb (*OR INPUT.bStorage_EstopPb*) OR StorageRobot_EStop OR ShippingRobot_EStop)  AND NOT EnableSimulation ;
E_StopEdgeDetect(xInput := Machine_Estop);
ResetEdgeDetect(xInput:= Machine_Reset);
StopEdgeDetect(xInput:= Machine_Stop);
StartEdgeDetect(xInput:= Machine_Start);

IF Allocate_EStopEdgeDetect.xRisingEdge THEN
	Allocate_EStop := FALSE;
ELSIF Allocate_EStopEdgeDetect.xFallingEdge THEN
	Allocate_EStop := TRUE;
END_IF

IF Storage_EstopEdgeDetect.xRisingEdge THEN
	Storage_EStop := FALSE;
ELSIF Storage_EstopEdgeDetect.xFallingEdge THEN
	Storage_EStop := TRUE;
END_IF

IF fbErrorHandler.ActiveAlarmCount <> 0 THEN
    xError := TRUE;
ELSE
    xError := FALSE;
END_IF

CASE fbErrorHandler.CurrentSeverityLevel OF
	E_Severity.Level7,E_Severity.Level6:
		IF xError AND (PackTag.Status.StateCurrent <> ePMLState_Aborted) THEN
			PackTag.Command.CntrlCmd := ePMLCommand_Abort;
		END_IF
END_CASE

IF ResetEdgeDetect.xRisingEdge THEN
//////////// Axis
	IF arAxisCtrl_gb[AxisNo.Allocate_X].Admin.Axis.Status.Error THEN
		arAxisCtrl_gb[AxisNo.Allocate_X].Admin.ClearError := Machine_Reset;
	END_IF
	IF arAxisCtrl_gb[AxisNo.Allocate_Y].Admin.Axis.Status.Error THEN
		arAxisCtrl_gb[AxisNo.Allocate_Y].Admin.ClearError := Machine_Reset;
	END_IF
	IF arAxisCtrl_gb[AxisNo.OutRobot_X].Admin.Axis.Status.Error THEN
		arAxisCtrl_gb[AxisNo.OutRobot_X].Admin.ClearError := Machine_Reset;
	END_IF
	IF arAxisCtrl_gb[AxisNo.OutRobot_Y].Admin.Axis.Status.Error THEN
		arAxisCtrl_gb[AxisNo.OutRobot_Y].Admin.ClearError := Machine_Reset;
	END_IF
	IF arAxisCtrl_gb[AxisNo.RoundBelt].Admin.Axis.Status.Error THEN
		arAxisCtrl_gb[AxisNo.RoundBelt].Admin.ClearError := Machine_Reset;
	END_IF
	IF arAxisCtrl_gb[AxisNo.TurnTable].Admin.Axis.Status.Error THEN
		arAxisCtrl_gb[AxisNo.TurnTable].Admin.ClearError := Machine_Reset;
	END_IF
	IF arAxisCtrl_gb[AxisNo.RackMotor].Admin.Axis.Status.Error THEN
		arAxisCtrl_gb[AxisNo.RackMotor].Admin.ClearError := Machine_Reset;
	END_IF
	
//////////// Cylinders
{region Cylinders }

